Staubli VAL3: Sychron_slave.dtx

bool bCycleOn
bool bRb2Home
bool bRb2InitOk
bool bRb2Ready
bool bRealM
bool bRes
bool bSetIO = true
bool bSychronOn
public bool bTest = true
bool bTxt1
bool bTxt2
bool bTxt3
bool bTxtPrSv = true
public bool bfnshint
bool ststu
dio fOut0 = {link=fOut0}
frame FrmDraw = {x=627.549581, y=-600.363481, z=-159.173811, rx=-90.113097, ry=-0.047506, rz=-0.047357, fatherId=world[0]}
jointRx jCad = {j1=15.222913, j2=48.613048, j3=81.686613, j4=179.999698, j5=130.298951, j6=-15.223398}
jointRx jConfig = {j1=-56.268773, j2=69.307617, j3=102.367275, j4=127.245004, j5=114.935336, j6=-7.907875}
jointRx jHome = {j1=-56.268773, j2=69.307617, j3=102.367275, j4=127.245004, j5=114.935336, j6=-7.907875}
jointRx jReal = {j1=15.453516, j2=48.799216, j3=80.615756, j4=179.999705, j5=129.41426, j6=-15.453992}
public mdesc mNomSpeed = {accel=30, decel=30, tmax=600, rmax=600, blend=off}
mdesc mSlow = {accel=30, decel=30, tmax=500, rmax=500}
num CmdTotal
num nDbg
num nPtTotal = 5
num nPulse[1500]
  [0] = 1
  [2] = 1
  [4] = 1
  [6] = 1
  [8] = 1
  [10] = 1
  [12] = 1
  [14] = 1
  [16] = 1
  [18] = 1
  [20] = 1
  [22] = 1
  [24] = 1
  [26] = 1
  [28] = 1
  [30] = 1
  [32] = 1
  [34] = 1
  [36] = 1
  [38] = 1
  [40] = 1
  [42] = 1
  [44] = 1
  [46] = 1
  [48] = 1
  [50] = 1
  [52] = 1
  [54] = 1
  [56] = 1
  [58] = 1
  [60] = 1
  [62] = 1
  [64] = 1
  [66] = 1
  [68] = 1
  [70] = 1
  [72] = 1
  [74] = 1
  [76] = 1
  [78] = 1
  [80] = 1
  [82] = 1
  [84] = 1
  [86] = 1
  [88] = 1
  [90] = 1
  [92] = 1
  [94] = 1
  [96] = 1
  [98] = 1
  [100] = 1
  [102] = 1
  [104] = 1
  [106] = 1
  [108] = 1
  [110] = 1
  [112] = 1
  [114] = 1
  [116] = 1
  [118] = 1
  [120] = 1
  [122] = 1
  [124] = 1
  [126] = 1
  [128] = 1
  [130] = 1
  [132] = 1
  [134] = 1
  [136] = 1
  [138] = 1
  [140] = 1
  [142] = 1
  [144] = 1
  [146] = 1
  [148] = 1
  [150] = 1
  [152] = 1
  [154] = 1
  [156] = 1
  [158] = 1
  [160] = 1
  [162] = 1
  [164] = 1
  [166] = 1
  [168] = 1
  [170] = 1
  [172] = 1
  [174] = 1
  [176] = 1
  [178] = 1
  [180] = 1
  [182] = 1
  [184] = 1
  [186] = 1
  [188] = 1
  [190] = 1
  [192] = 1
  [194] = 1
  [196] = 1
  [198] = 1
  [200] = 1
  [202] = 1
  [204] = 1
  [206] = 1
  [208] = 1
  [210] = 1
  [212] = 1
  [214] = 1
  [216] = 1
  [218] = 1
  [220] = 1
  [222] = 1
  [224] = 1
  [226] = 1
  [228] = 1
  [230] = 1
  [232] = 1
  [234] = 1
  [236] = 1
  [238] = 1
  [240] = 1
  [242] = 1
  [244] = 1
  [246] = 1
  [248] = 1
  [250] = 1
  [252] = 1
  [254] = 1
  [256] = 1
  [258] = 1
  [260] = 1
  [262] = 1
  [264] = 1
  [266] = 1
  [268] = 1
  [270] = 1
  [272] = 1
  [274] = 1
  [276] = 1
  [278] = 1
  [280] = 1
  [282] = 1
  [284] = 1
  [286] = 1
  [288] = 1
  [290] = 1
  [292] = 1
  [294] = 1
  [296] = 1
  [298] = 1
  [300] = 1
  [302] = 1
  [304] = 1
  [306] = 1
  [308] = 1
  [310] = 1
  [312] = 1
  [314] = 1
  [316] = 1
  [318] = 1
  [320] = 1
  [322] = 1
  [324] = 1
  [326] = 1
  [328] = 1
  [330] = 1
  [332] = 1
  [334] = 1
  [336] = 1
  [338] = 1
  [340] = 1
  [342] = 1
  [344] = 1
  [346] = 1
  [348] = 1
  [350] = 1
  [352] = 1
  [354] = 1
  [356] = 1
  [358] = 1
  [360] = 1
  [362] = 1
  [364] = 1
  [366] = 1
  [368] = 1
  [370] = 1
  [372] = 1
  [374] = 1
  [376] = 1
  [378] = 1
  [380] = 1
  [382] = 1
  [384] = 1
  [386] = 1
  [388] = 1
  [390] = 1
  [392] = 1
  [394] = 1
  [396] = 1
  [398] = 1
  [400] = 1
  [402] = 1
  [404] = 1
  [406] = 1
  [408] = 1
  [410] = 1
  [412] = 1
  [414] = 1
  [416] = 1
  [418] = 1
  [420] = 1
  [422] = 1
  [424] = 1
  [426] = 1
  [428] = 1
  [430] = 1
  [432] = 1
  [434] = 1
  [436] = 1
  [438] = 1
  [440] = 1
  [442] = 1
  [444] = 1
  [446] = 1
  [448] = 1
  [450] = 1
  [452] = 1
  [454] = 1
  [456] = 1
  [458] = 1
  [460] = 1
  [462] = 1
  [464] = 1
  [466] = 1
  [468] = 1
  [470] = 1
  [472] = 1
  [474] = 1
  [476] = 1
  [478] = 1
  [480] = 1
  [482] = 1
  [484] = 1
  [486] = 1
  [488] = 1
  [490] = 1
  [492] = 1
  [494] = 1
  [496] = 1
  [498] = 1
  [500] = 1
  [502] = 1
  [504] = 1
  [506] = 1
  [508] = 1
  [510] = 1
  [512] = 1
  [514] = 1
  [516] = 1
  [518] = 1
  [520] = 1
  [522] = 1
  [524] = 1
  [526] = 1
  [528] = 1
  [530] = 1
  [532] = 1
  [534] = 1
  [536] = 1
  [538] = 1
  [540] = 1
  [542] = 1
  [544] = 1
  [546] = 1
  [548] = 1
  [550] = 1
  [552] = 1
  [554] = 1
  [556] = 1
  [558] = 1
  [560] = 1
  [562] = 1
  [564] = 1
  [566] = 1
  [568] = 1
  [570] = 1
  [572] = 1
  [574] = 1
  [576] = 1
  [578] = 1
  [580] = 1
  [582] = 1
  [584] = 1
  [586] = 1
  [588] = 1
  [590] = 1
  [592] = 1
  [594] = 1
  [596] = 1
  [598] = 1
  [600] = 1
  [602] = 1
  [604] = 1
  [606] = 1
  [608] = 1
  [610] = 1
  [612] = 1
  [614] = 1
  [616] = 1
  [618] = 1
  [620] = 1
  [622] = 1
  [624] = 1
  [626] = 1
  [628] = 1
  [630] = 1
  [632] = 1
  [634] = 1
  [636] = 1
  [638] = 1
  [640] = 1
  [642] = 1
  [644] = 1
  [646] = 1
  [648] = 1
  [650] = 1
  [652] = 1
  [654] = 1
  [656] = 1
  [658] = 1
  [660] = 1
  [662] = 1
  [664] = 1
  [666] = 1
  [668] = 1
  [670] = 1
  [672] = 1
  [674] = 1
  [676] = 1
  [678] = 1
  [680] = 1
  [682] = 1
  [684] = 1
  [686] = 1
  [688] = 1
  [690] = 1
  [692] = 1
  [694] = 1
  [696] = 1
  [698] = 1
  [700] = 1
  [702] = 1
  [704] = 1
  [706] = 1
  [708] = 1
  [710] = 1
  [712] = 1
  [714] = 1
  [716] = 1
  [718] = 1
  [720] = 1
  [722] = 1
  [724] = 1
  [726] = 1
  [728] = 1
  [730] = 1
  [732] = 1
  [734] = 1
  [736] = 1
  [738] = 1
  [740] = 1
  [742] = 1
  [744] = 1
  [746] = 1
  [748] = 1
  [750] = 1
  [752] = 1
  [754] = 1
  [756] = 1
  [758] = 1
  [760] = 1
  [762] = 1
  [764] = 1
  [766] = 1
  [768] = 1
  [770] = 1
  [772] = 1
  [774] = 1
  [776] = 1
  [778] = 1
  [780] = 1
  [782] = 1
  [784] = 1
  [786] = 1
  [788] = 1
  [790] = 1
  [792] = 1
  [794] = 1
  [796] = 1
  [798] = 1
  [800] = 1
  [802] = 1
  [804] = 1
  [806] = 1
  [808] = 1
  [810] = 1
  [812] = 1
  [814] = 1
  [816] = 1
  [818] = 1
  [820] = 1
  [822] = 1
  [824] = 1
  [826] = 1
  [828] = 1
  [830] = 1
  [832] = 1
  [834] = 1
  [836] = 1
  [838] = 1
  [840] = 1
  [842] = 1
  [844] = 1
  [846] = 1
  [848] = 1
  [850] = 1
  [852] = 1
  [854] = 1
  [856] = 1
  [858] = 1
  [860] = 1
  [862] = 1
  [864] = 1
  [866] = 1
  [868] = 1
  [870] = 1
  [872] = 1
  [874] = 1
  [876] = 1
  [878] = 1
  [880] = 1
  [882] = 1
  [884] = 1
  [886] = 1
  [888] = 1
  [890] = 1
  [892] = 1
  [894] = 1
  [896] = 1
  [898] = 1
  [900] = 1
  [902] = 1
  [904] = 1
  [906] = 1
  [908] = 1
  [910] = 1
  [912] = 1
  [914] = 1
  [916] = 1
  [918] = 1
  [920] = 1
  [922] = 1
  [924] = 1
  [926] = 1
  [928] = 1
  [930] = 1
  [932] = 1
  [934] = 1
  [936] = 1
  [938] = 1
  [940] = 1
  [942] = 1
  [944] = 1
  [946] = 1
  [948] = 1
  [950] = 1
  [952] = 1
  [954] = 1
  [956] = 1
  [958] = 1
  [960] = 1
  [962] = 1
  [964] = 1
  [966] = 1
  [968] = 1
  [970] = 1
  [972] = 1
  [974] = 1
  [976] = 1
  [978] = 1
  [980] = 1
  [982] = 1
  [984] = 1
  [986] = 1
  [988] = 1
  [990] = 1
  [992] = 1
  [994] = 1
  [996] = 1
  [998] = 1
num nReadPt
num nScrPts = 1291
public num nTestNum = 2
public num nTime = 0.001
num nTotalPoints = 1
num nTxtTotal = 347
num nWritePt
num n_sTxt = 2
num nn = 3048
num nsumtime = 5916.439
pointRx MoveTo = {ry=-90, rz=174.889504, fatherId=FrmDraw[0]}
pointRx Zero = {ry=-90, rz=174.889504, fatherId=FrmDraw[0]}
pointRx frm_ori = {x=627.549581, y=-600.363481, z=-159.173811, ry=90, rz=179.586129, fatherId=world[0]}
pointRx frm_x = {x=876.01171, y=-600.157069, z=-158.968855, rx=4.422019, ry=89.999088, rz=175.164786, fatherId=world[0]}
pointRx frm_y = {x=875.958066, y=-600.377284, z=-270.508394, ry=90, rz=179.586975, fatherId=world[0]}
pointRx pChange = {fatherId=FrmDraw[0]}
pointRx pfrmCad[1500]
  [0] = {x=52.63, y=-161.79, z=1, rx=-90, ry=53.98, fatherId=FrmDraw[0]}
  [1] = {x=52.51, y=-161.63, z=1, rx=-90, ry=54, fatherId=FrmDraw[0]}
  [2] = {x=52.39, y=-161.46, z=1, rx=-90, ry=54.05, fatherId=FrmDraw[0]}
  [3] = {x=52.27, y=-161.3, z=1, rx=-90, ry=54.09, fatherId=FrmDraw[0]}
  [4] = {x=52.16, y=-161.14, z=1, rx=-90, ry=54.13, fatherId=FrmDraw[0]}
  [5] = {x=52.04, y=-160.98, z=1, rx=-90, ry=54.17, fatherId=FrmDraw[0]}
  [6] = {x=51.92, y=-160.82, z=1, rx=-90, ry=54.21, fatherId=FrmDraw[0]}
  [7] = {x=51.81, y=-160.65, z=1, rx=-90, ry=54.25, fatherId=FrmDraw[0]}
  [8] = {x=51.69, y=-160.49, z=1, rx=-90, ry=54.3, fatherId=FrmDraw[0]}
  [9] = {x=51.57, y=-160.33, z=1, rx=-90, ry=54.34, fatherId=FrmDraw[0]}
  [10] = {x=51.46, y=-160.17, z=1, rx=-90, ry=54.38, fatherId=FrmDraw[0]}
  [11] = {x=51.34, y=-160, z=1, rx=-90, ry=54.42, fatherId=FrmDraw[0]}
  [12] = {x=51.22, y=-159.84, z=1, rx=-90, ry=54.46, fatherId=FrmDraw[0]}
  [13] = {x=51.11, y=-159.68, z=1, rx=-90, ry=54.5, fatherId=FrmDraw[0]}
  [14] = {x=50.99, y=-159.52, z=1, rx=-90, ry=54.55, fatherId=FrmDraw[0]}
  [15] = {x=50.88, y=-159.35, z=1, rx=-90, ry=54.59, fatherId=FrmDraw[0]}
  [16] = {x=50.76, y=-159.19, z=1, rx=-90, ry=54.63, fatherId=FrmDraw[0]}
  [17] = {x=50.64, y=-159.03, z=1, rx=-90, ry=54.67, fatherId=FrmDraw[0]}
  [18] = {x=50.53, y=-158.86, z=1, rx=-90, ry=54.71, fatherId=FrmDraw[0]}
  [19] = {x=50.41, y=-158.7, z=1, rx=-90, ry=54.75, fatherId=FrmDraw[0]}
  [20] = {x=50.3, y=-158.54, z=1, rx=-90, ry=54.8, fatherId=FrmDraw[0]}
  [21] = {x=50.18, y=-158.37, z=1, rx=-90, ry=54.84, fatherId=FrmDraw[0]}
  [22] = {x=50.07, y=-158.21, z=1, rx=-90, ry=54.88, fatherId=FrmDraw[0]}
  [23] = {x=49.95, y=-158.05, z=1, rx=-90, ry=54.92, fatherId=FrmDraw[0]}
  [24] = {x=49.84, y=-157.88, z=1, rx=-90, ry=54.96, fatherId=FrmDraw[0]}
  [25] = {x=49.72, y=-157.72, z=1, rx=-90, ry=55, fatherId=FrmDraw[0]}
  [26] = {x=49.61, y=-157.55, z=1, rx=-90, ry=55.05, fatherId=FrmDraw[0]}
  [27] = {x=49.49, y=-157.39, z=1, rx=-90, ry=55.09, fatherId=FrmDraw[0]}
  [28] = {x=49.38, y=-157.23, z=1, rx=-90, ry=55.13, fatherId=FrmDraw[0]}
  [29] = {x=49.26, y=-157.06, z=1, rx=-90, ry=55.17, fatherId=FrmDraw[0]}
  [30] = {x=49.15, y=-156.9, z=1, rx=-90, ry=55.21, fatherId=FrmDraw[0]}
  [31] = {x=49.04, y=-156.73, z=1, rx=-90, ry=55.25, fatherId=FrmDraw[0]}
  [32] = {x=48.92, y=-156.57, z=1, rx=-90, ry=55.3, fatherId=FrmDraw[0]}
  [33] = {x=48.81, y=-156.4, z=1, rx=-90, ry=55.34, fatherId=FrmDraw[0]}
  [34] = {x=48.69, y=-156.24, z=1, rx=-90, ry=55.38, fatherId=FrmDraw[0]}
  [35] = {x=48.58, y=-156.08, z=1, rx=-90, ry=55.42, fatherId=FrmDraw[0]}
  [36] = {x=48.47, y=-155.91, z=1, rx=-90, ry=55.46, fatherId=FrmDraw[0]}
  [37] = {x=48.35, y=-155.75, z=1, rx=-90, ry=55.5, fatherId=FrmDraw[0]}
  [38] = {x=48.24, y=-155.58, z=1, rx=-90, ry=55.55, fatherId=FrmDraw[0]}
  [39] = {x=48.13, y=-155.42, z=1, rx=-90, ry=55.59, fatherId=FrmDraw[0]}
  [40] = {x=48.02, y=-155.25, z=1, rx=-90, ry=55.63, fatherId=FrmDraw[0]}
  [41] = {x=47.9, y=-155.09, z=1, rx=-90, ry=55.67, fatherId=FrmDraw[0]}
  [42] = {x=47.79, y=-154.92, z=1, rx=-90, ry=55.71, fatherId=FrmDraw[0]}
  [43] = {x=47.68, y=-154.76, z=1, rx=-90, ry=55.75, fatherId=FrmDraw[0]}
  [44] = {x=47.56, y=-154.59, z=1, rx=-90, ry=55.8, fatherId=FrmDraw[0]}
  [45] = {x=47.45, y=-154.42, z=1, rx=-90, ry=55.84, fatherId=FrmDraw[0]}
  [46] = {x=47.34, y=-154.26, z=1, rx=-90, ry=55.88, fatherId=FrmDraw[0]}
  [47] = {x=47.23, y=-154.09, z=1, rx=-90, ry=55.92, fatherId=FrmDraw[0]}
  [48] = {x=47.12, y=-153.93, z=1, rx=-90, ry=55.96, fatherId=FrmDraw[0]}
  [49] = {x=47, y=-153.76, z=1, rx=-90, ry=56, fatherId=FrmDraw[0]}
  [50] = {x=46.89, y=-153.6, z=1, rx=-90, ry=56.05, fatherId=FrmDraw[0]}
  [51] = {x=46.78, y=-153.43, z=1, rx=-90, ry=56.09, fatherId=FrmDraw[0]}
  [52] = {x=46.67, y=-153.26, z=1, rx=-90, ry=56.13, fatherId=FrmDraw[0]}
  [53] = {x=46.56, y=-153.1, z=1, rx=-90, ry=56.17, fatherId=FrmDraw[0]}
  [54] = {x=46.45, y=-152.93, z=1, rx=-90, ry=56.21, fatherId=FrmDraw[0]}
  [55] = {x=46.34, y=-152.77, z=1, rx=-90, ry=56.25, fatherId=FrmDraw[0]}
  [56] = {x=46.22, y=-152.6, z=1, rx=-90, ry=56.3, fatherId=FrmDraw[0]}
  [57] = {x=46.11, y=-152.43, z=1, rx=-90, ry=56.34, fatherId=FrmDraw[0]}
  [58] = {x=46, y=-152.27, z=1, rx=-90, ry=56.38, fatherId=FrmDraw[0]}
  [59] = {x=45.89, y=-152.1, z=1, rx=-90, ry=56.42, fatherId=FrmDraw[0]}
  [60] = {x=45.78, y=-151.93, z=1, rx=-90, ry=56.46, fatherId=FrmDraw[0]}
  [61] = {x=45.67, y=-151.77, z=1, rx=-90, ry=56.5, fatherId=FrmDraw[0]}
  [62] = {x=45.56, y=-151.6, z=1, rx=-90, ry=56.55, fatherId=FrmDraw[0]}
  [63] = {x=45.45, y=-151.43, z=1, rx=-90, ry=56.59, fatherId=FrmDraw[0]}
  [64] = {x=45.34, y=-151.27, z=1, rx=-90, ry=56.63, fatherId=FrmDraw[0]}
  [65] = {x=45.23, y=-151.1, z=1, rx=-90, ry=56.67, fatherId=FrmDraw[0]}
  [66] = {x=45.12, y=-150.93, z=1, rx=-90, ry=56.71, fatherId=FrmDraw[0]}
  [67] = {x=45.01, y=-150.76, z=1, rx=-90, ry=56.75, fatherId=FrmDraw[0]}
  [68] = {x=44.9, y=-150.6, z=1, rx=-90, ry=56.8, fatherId=FrmDraw[0]}
  [69] = {x=44.79, y=-150.43, z=1, rx=-90, ry=56.84, fatherId=FrmDraw[0]}
  [70] = {x=44.68, y=-150.26, z=1, rx=-90, ry=56.88, fatherId=FrmDraw[0]}
  [71] = {x=44.57, y=-150.09, z=1, rx=-90, ry=56.92, fatherId=FrmDraw[0]}
  [72] = {x=44.46, y=-149.93, z=1, rx=-90, ry=56.96, fatherId=FrmDraw[0]}
  [73] = {x=44.35, y=-149.76, z=1, rx=-90, ry=57, fatherId=FrmDraw[0]}
  [74] = {x=44.25, y=-149.59, z=1, rx=-90, ry=57.05, fatherId=FrmDraw[0]}
  [75] = {x=44.14, y=-149.42, z=1, rx=-90, ry=57.09, fatherId=FrmDraw[0]}
  [76] = {x=44.03, y=-149.26, z=1, rx=-90, ry=57.13, fatherId=FrmDraw[0]}
  [77] = {x=43.92, y=-149.09, z=1, rx=-90, ry=57.17, fatherId=FrmDraw[0]}
  [78] = {x=43.81, y=-148.92, z=1, rx=-90, ry=57.21, fatherId=FrmDraw[0]}
  [79] = {x=43.7, y=-148.75, z=1, rx=-90, ry=57.25, fatherId=FrmDraw[0]}
  [80] = {x=43.6, y=-148.58, z=1, rx=-90, ry=57.3, fatherId=FrmDraw[0]}
  [81] = {x=43.49, y=-148.41, z=1, rx=-90, ry=57.34, fatherId=FrmDraw[0]}
  [82] = {x=43.38, y=-148.25, z=1, rx=-90, ry=57.38, fatherId=FrmDraw[0]}
  [83] = {x=43.27, y=-148.08, z=1, rx=-90, ry=57.42, fatherId=FrmDraw[0]}
  [84] = {x=43.16, y=-147.91, z=1, rx=-90, ry=57.46, fatherId=FrmDraw[0]}
  [85] = {x=43.06, y=-147.74, z=1, rx=-90, ry=57.5, fatherId=FrmDraw[0]}
  [86] = {x=42.95, y=-147.57, z=1, rx=-90, ry=57.55, fatherId=FrmDraw[0]}
  [87] = {x=42.84, y=-147.4, z=1, rx=-90, ry=57.59, fatherId=FrmDraw[0]}
  [88] = {x=42.73, y=-147.23, z=1, rx=-90, ry=57.63, fatherId=FrmDraw[0]}
  [89] = {x=42.63, y=-147.07, z=1, rx=-90, ry=57.67, fatherId=FrmDraw[0]}
  [90] = {x=42.52, y=-146.9, z=1, rx=-90, ry=57.71, fatherId=FrmDraw[0]}
  [91] = {x=42.41, y=-146.73, z=1, rx=-90, ry=57.75, fatherId=FrmDraw[0]}
  [92] = {x=42.31, y=-146.56, z=1, rx=-90, ry=57.8, fatherId=FrmDraw[0]}
  [93] = {x=42.2, y=-146.39, z=1, rx=-90, ry=57.84, fatherId=FrmDraw[0]}
  [94] = {x=42.09, y=-146.22, z=1, rx=-90, ry=57.88, fatherId=FrmDraw[0]}
  [95] = {x=41.99, y=-146.05, z=1, rx=-90, ry=57.92, fatherId=FrmDraw[0]}
  [96] = {x=41.88, y=-145.88, z=1, rx=-90, ry=57.96, fatherId=FrmDraw[0]}
  [97] = {x=41.78, y=-145.71, z=1, rx=-90, ry=58, fatherId=FrmDraw[0]}
  [98] = {x=41.67, y=-145.54, z=1, rx=-90, ry=58.05, fatherId=FrmDraw[0]}
  [99] = {x=41.56, y=-145.37, z=1, rx=-90, ry=58.09, fatherId=FrmDraw[0]}
  [100] = {x=41.46, y=-145.2, z=1, rx=-90, ry=58.13, fatherId=FrmDraw[0]}
  [101] = {x=41.35, y=-145.03, z=1, rx=-90, ry=58.17, fatherId=FrmDraw[0]}
  [102] = {x=41.25, y=-144.86, z=1, rx=-90, ry=58.21, fatherId=FrmDraw[0]}
  [103] = {x=41.14, y=-144.69, z=1, rx=-90, ry=58.25, fatherId=FrmDraw[0]}
  [104] = {x=41.04, y=-144.52, z=1, rx=-90, ry=58.3, fatherId=FrmDraw[0]}
  [105] = {x=40.93, y=-144.35, z=1, rx=-90, ry=58.34, fatherId=FrmDraw[0]}
  [106] = {x=40.83, y=-144.18, z=1, rx=-90, ry=58.38, fatherId=FrmDraw[0]}
  [107] = {x=40.72, y=-144.01, z=1, rx=-90, ry=58.42, fatherId=FrmDraw[0]}
  [108] = {x=40.62, y=-143.84, z=1, rx=-90, ry=58.46, fatherId=FrmDraw[0]}
  [109] = {x=40.51, y=-143.67, z=1, rx=-90, ry=58.5, fatherId=FrmDraw[0]}
  [110] = {x=40.41, y=-143.5, z=1, rx=-90, ry=58.55, fatherId=FrmDraw[0]}
  [111] = {x=40.3, y=-143.33, z=1, rx=-90, ry=58.59, fatherId=FrmDraw[0]}
  [112] = {x=40.2, y=-143.16, z=1, rx=-90, ry=58.63, fatherId=FrmDraw[0]}
  [113] = {x=40.1, y=-142.99, z=1, rx=-90, ry=58.67, fatherId=FrmDraw[0]}
  [114] = {x=39.99, y=-142.82, z=1, rx=-90, ry=58.71, fatherId=FrmDraw[0]}
  [115] = {x=39.89, y=-142.65, z=1, rx=-90, ry=58.75, fatherId=FrmDraw[0]}
  [116] = {x=39.79, y=-142.47, z=1, rx=-90, ry=58.8, fatherId=FrmDraw[0]}
  [117] = {x=39.68, y=-142.3, z=1, rx=-90, ry=58.84, fatherId=FrmDraw[0]}
  [118] = {x=39.58, y=-142.13, z=1, rx=-90, ry=58.88, fatherId=FrmDraw[0]}
  [119] = {x=39.47, y=-141.96, z=1, rx=-90, ry=58.92, fatherId=FrmDraw[0]}
  [120] = {x=39.37, y=-141.79, z=1, rx=-90, ry=58.96, fatherId=FrmDraw[0]}
  [121] = {x=39.27, y=-141.62, z=1, rx=-90, ry=59, fatherId=FrmDraw[0]}
  [122] = {x=39.17, y=-141.45, z=1, rx=-90, ry=59.05, fatherId=FrmDraw[0]}
  [123] = {x=39.06, y=-141.28, z=1, rx=-90, ry=59.09, fatherId=FrmDraw[0]}
  [124] = {x=38.96, y=-141.1, z=1, rx=-90, ry=59.13, fatherId=FrmDraw[0]}
  [125] = {x=38.86, y=-140.93, z=1, rx=-90, ry=59.17, fatherId=FrmDraw[0]}
  [126] = {x=38.76, y=-140.76, z=1, rx=-90, ry=59.21, fatherId=FrmDraw[0]}
  [127] = {x=38.65, y=-140.59, z=1, rx=-90, ry=59.25, fatherId=FrmDraw[0]}
  [128] = {x=38.55, y=-140.42, z=1, rx=-90, ry=59.3, fatherId=FrmDraw[0]}
  [129] = {x=38.45, y=-140.24, z=1, rx=-90, ry=59.34, fatherId=FrmDraw[0]}
  [130] = {x=38.35, y=-140.07, z=1, rx=-90, ry=59.38, fatherId=FrmDraw[0]}
  [131] = {x=38.24, y=-139.9, z=1, rx=-90, ry=59.42, fatherId=FrmDraw[0]}
  [132] = {x=38.14, y=-139.73, z=1, rx=-90, ry=59.46, fatherId=FrmDraw[0]}
  [133] = {x=38.04, y=-139.56, z=1, rx=-90, ry=59.5, fatherId=FrmDraw[0]}
  [134] = {x=37.94, y=-139.38, z=1, rx=-90, ry=59.55, fatherId=FrmDraw[0]}
  [135] = {x=37.84, y=-139.21, z=1, rx=-90, ry=59.59, fatherId=FrmDraw[0]}
  [136] = {x=37.74, y=-139.04, z=1, rx=-90, ry=59.63, fatherId=FrmDraw[0]}
  [137] = {x=37.64, y=-138.87, z=1, rx=-90, ry=59.67, fatherId=FrmDraw[0]}
  [138] = {x=37.54, y=-138.69, z=1, rx=-90, ry=59.71, fatherId=FrmDraw[0]}
  [139] = {x=37.43, y=-138.52, z=1, rx=-90, ry=59.75, fatherId=FrmDraw[0]}
  [140] = {x=37.33, y=-138.35, z=1, rx=-90, ry=59.8, fatherId=FrmDraw[0]}
  [141] = {x=37.23, y=-138.17, z=1, rx=-90, ry=59.84, fatherId=FrmDraw[0]}
  [142] = {x=37.13, y=-138, z=1, rx=-90, ry=59.88, fatherId=FrmDraw[0]}
  [143] = {x=37.03, y=-137.83, z=1, rx=-90, ry=59.92, fatherId=FrmDraw[0]}
  [144] = {x=36.93, y=-137.66, z=1, rx=-90, ry=59.96, fatherId=FrmDraw[0]}
  [145] = {x=36.83, y=-137.48, z=1, rx=-90, ry=60, fatherId=FrmDraw[0]}
  [146] = {x=36.73, y=-137.31, z=1, rx=-90, ry=60.05, fatherId=FrmDraw[0]}
  [147] = {x=36.63, y=-137.14, z=1, rx=-90, ry=60.09, fatherId=FrmDraw[0]}
  [148] = {x=36.53, y=-136.96, z=1, rx=-90, ry=60.13, fatherId=FrmDraw[0]}
  [149] = {x=36.43, y=-136.79, z=1, rx=-90, ry=60.17, fatherId=FrmDraw[0]}
  [150] = {x=36.33, y=-136.62, z=1, rx=-90, ry=60.21, fatherId=FrmDraw[0]}
  [151] = {x=36.24, y=-136.44, z=1, rx=-90, ry=60.25, fatherId=FrmDraw[0]}
  [152] = {x=36.14, y=-136.27, z=1, rx=-90, ry=60.3, fatherId=FrmDraw[0]}
  [153] = {x=36.04, y=-136.09, z=1, rx=-90, ry=60.34, fatherId=FrmDraw[0]}
  [154] = {x=35.94, y=-135.92, z=1, rx=-90, ry=60.38, fatherId=FrmDraw[0]}
  [155] = {x=35.84, y=-135.75, z=1, rx=-90, ry=60.42, fatherId=FrmDraw[0]}
  [156] = {x=35.74, y=-135.57, z=1, rx=-90, ry=60.46, fatherId=FrmDraw[0]}
  [157] = {x=35.64, y=-135.4, z=1, rx=-90, ry=60.5, fatherId=FrmDraw[0]}
  [158] = {x=35.54, y=-135.22, z=1, rx=-90, ry=60.55, fatherId=FrmDraw[0]}
  [159] = {x=35.45, y=-135.05, z=1, rx=-90, ry=60.59, fatherId=FrmDraw[0]}
  [160] = {x=35.35, y=-134.88, z=1, rx=-90, ry=60.63, fatherId=FrmDraw[0]}
  [161] = {x=35.25, y=-134.7, z=1, rx=-90, ry=60.67, fatherId=FrmDraw[0]}
  [162] = {x=35.15, y=-134.53, z=1, rx=-90, ry=60.71, fatherId=FrmDraw[0]}
  [163] = {x=35.05, y=-134.35, z=1, rx=-90, ry=60.75, fatherId=FrmDraw[0]}
  [164] = {x=34.96, y=-134.18, z=1, rx=-90, ry=60.8, fatherId=FrmDraw[0]}
  [165] = {x=34.86, y=-134, z=1, rx=-90, ry=60.84, fatherId=FrmDraw[0]}
  [166] = {x=34.76, y=-133.83, z=1, rx=-90, ry=60.88, fatherId=FrmDraw[0]}
  [167] = {x=34.66, y=-133.65, z=1, rx=-90, ry=60.92, fatherId=FrmDraw[0]}
  [168] = {x=34.57, y=-133.48, z=1, rx=-90, ry=60.96, fatherId=FrmDraw[0]}
  [169] = {x=34.47, y=-133.3, z=1, rx=-90, ry=61, fatherId=FrmDraw[0]}
  [170] = {x=34.37, y=-133.13, z=1, rx=-90, ry=61.05, fatherId=FrmDraw[0]}
  [171] = {x=34.28, y=-132.95, z=1, rx=-90, ry=61.09, fatherId=FrmDraw[0]}
  [172] = {x=34.18, y=-132.78, z=1, rx=-90, ry=61.13, fatherId=FrmDraw[0]}
  [173] = {x=34.08, y=-132.6, z=1, rx=-90, ry=61.17, fatherId=FrmDraw[0]}
  [174] = {x=33.99, y=-132.43, z=1, rx=-90, ry=61.21, fatherId=FrmDraw[0]}
  [175] = {x=33.89, y=-132.25, z=1, rx=-90, ry=61.25, fatherId=FrmDraw[0]}
  [176] = {x=33.79, y=-132.08, z=1, rx=-90, ry=61.3, fatherId=FrmDraw[0]}
  [177] = {x=33.7, y=-131.9, z=1, rx=-90, ry=61.34, fatherId=FrmDraw[0]}
  [178] = {x=33.6, y=-131.73, z=1, rx=-90, ry=61.38, fatherId=FrmDraw[0]}
  [179] = {x=33.51, y=-131.55, z=1, rx=-90, ry=61.42, fatherId=FrmDraw[0]}
  [180] = {x=33.41, y=-131.38, z=1, rx=-90, ry=61.46, fatherId=FrmDraw[0]}
  [181] = {x=33.32, y=-131.2, z=1, rx=-90, ry=61.5, fatherId=FrmDraw[0]}
  [182] = {x=33.22, y=-131.02, z=1, rx=-90, ry=61.55, fatherId=FrmDraw[0]}
  [183] = {x=33.12, y=-130.85, z=1, rx=-90, ry=61.59, fatherId=FrmDraw[0]}
  [184] = {x=33.03, y=-130.67, z=1, rx=-90, ry=61.63, fatherId=FrmDraw[0]}
  [185] = {x=32.93, y=-130.5, z=1, rx=-90, ry=61.67, fatherId=FrmDraw[0]}
  [186] = {x=32.84, y=-130.32, z=1, rx=-90, ry=61.71, fatherId=FrmDraw[0]}
  [187] = {x=32.74, y=-130.14, z=1, rx=-90, ry=61.75, fatherId=FrmDraw[0]}
  [188] = {x=32.65, y=-129.97, z=1, rx=-90, ry=61.8, fatherId=FrmDraw[0]}
  [189] = {x=32.56, y=-129.79, z=1, rx=-90, ry=61.84, fatherId=FrmDraw[0]}
  [190] = {x=32.46, y=-129.62, z=1, rx=-90, ry=61.88, fatherId=FrmDraw[0]}
  [191] = {x=32.37, y=-129.44, z=1, rx=-90, ry=61.92, fatherId=FrmDraw[0]}
  [192] = {x=32.27, y=-129.26, z=1, rx=-90, ry=61.96, fatherId=FrmDraw[0]}
  [193] = {x=32.18, y=-129.09, z=1, rx=-90, ry=62, fatherId=FrmDraw[0]}
  [194] = {x=32.09, y=-128.91, z=1, rx=-90, ry=62.05, fatherId=FrmDraw[0]}
  [195] = {x=31.99, y=-128.73, z=1, rx=-90, ry=62.09, fatherId=FrmDraw[0]}
  [196] = {x=31.9, y=-128.56, z=1, rx=-90, ry=62.13, fatherId=FrmDraw[0]}
  [197] = {x=31.8, y=-128.38, z=1, rx=-90, ry=62.17, fatherId=FrmDraw[0]}
  [198] = {x=31.71, y=-128.2, z=1, rx=-90, ry=62.21, fatherId=FrmDraw[0]}
  [199] = {x=31.62, y=-128.03, z=1, rx=-90, ry=62.25, fatherId=FrmDraw[0]}
  [200] = {x=31.53, y=-127.85, z=1, rx=-90, ry=62.3, fatherId=FrmDraw[0]}
  [201] = {x=31.43, y=-127.67, z=1, rx=-90, ry=62.34, fatherId=FrmDraw[0]}
  [202] = {x=31.34, y=-127.49, z=1, rx=-90, ry=62.38, fatherId=FrmDraw[0]}
  [203] = {x=31.25, y=-127.32, z=1, rx=-90, ry=62.42, fatherId=FrmDraw[0]}
  [204] = {x=31.15, y=-127.14, z=1, rx=-90, ry=62.46, fatherId=FrmDraw[0]}
  [205] = {x=31.06, y=-126.96, z=1, rx=-90, ry=62.5, fatherId=FrmDraw[0]}
  [206] = {x=30.97, y=-126.78, z=1, rx=-90, ry=62.55, fatherId=FrmDraw[0]}
  [207] = {x=30.88, y=-126.61, z=1, rx=-90, ry=62.59, fatherId=FrmDraw[0]}
  [208] = {x=30.79, y=-126.43, z=1, rx=-90, ry=62.63, fatherId=FrmDraw[0]}
  [209] = {x=30.69, y=-126.25, z=1, rx=-90, ry=62.67, fatherId=FrmDraw[0]}
  [210] = {x=30.6, y=-126.07, z=1, rx=-90, ry=62.71, fatherId=FrmDraw[0]}
  [211] = {x=30.51, y=-125.9, z=1, rx=-90, ry=62.75, fatherId=FrmDraw[0]}
  [212] = {x=30.42, y=-125.72, z=1, rx=-90, ry=62.8, fatherId=FrmDraw[0]}
  [213] = {x=30.33, y=-125.54, z=1, rx=-90, ry=62.84, fatherId=FrmDraw[0]}
  [214] = {x=30.24, y=-125.36, z=1, rx=-90, ry=62.88, fatherId=FrmDraw[0]}
  [215] = {x=30.15, y=-125.18, z=1, rx=-90, ry=62.92, fatherId=FrmDraw[0]}
  [216] = {x=30.05, y=-125.01, z=1, rx=-90, ry=62.96, fatherId=FrmDraw[0]}
  [217] = {x=29.96, y=-124.83, z=1, rx=-90, ry=63, fatherId=FrmDraw[0]}
  [218] = {x=29.87, y=-124.65, z=1, rx=-90, ry=63.05, fatherId=FrmDraw[0]}
  [219] = {x=29.78, y=-124.47, z=1, rx=-90, ry=63.09, fatherId=FrmDraw[0]}
  [220] = {x=29.69, y=-124.29, z=1, rx=-90, ry=63.13, fatherId=FrmDraw[0]}
  [221] = {x=29.6, y=-124.11, z=1, rx=-90, ry=63.17, fatherId=FrmDraw[0]}
  [222] = {x=29.51, y=-123.94, z=1, rx=-90, ry=63.21, fatherId=FrmDraw[0]}
  [223] = {x=29.42, y=-123.76, z=1, rx=-90, ry=63.25, fatherId=FrmDraw[0]}
  [224] = {x=29.33, y=-123.58, z=1, rx=-90, ry=63.3, fatherId=FrmDraw[0]}
  [225] = {x=29.24, y=-123.4, z=1, rx=-90, ry=63.34, fatherId=FrmDraw[0]}
  [226] = {x=29.15, y=-123.22, z=1, rx=-90, ry=63.38, fatherId=FrmDraw[0]}
  [227] = {x=29.06, y=-123.04, z=1, rx=-90, ry=63.42, fatherId=FrmDraw[0]}
  [228] = {x=28.97, y=-122.86, z=1, rx=-90, ry=63.46, fatherId=FrmDraw[0]}
  [229] = {x=28.88, y=-122.68, z=1, rx=-90, ry=63.5, fatherId=FrmDraw[0]}
  [230] = {x=28.79, y=-122.51, z=1, rx=-90, ry=63.55, fatherId=FrmDraw[0]}
  [231] = {x=28.71, y=-122.33, z=1, rx=-90, ry=63.59, fatherId=FrmDraw[0]}
  [232] = {x=28.62, y=-122.15, z=1, rx=-90, ry=63.63, fatherId=FrmDraw[0]}
  [233] = {x=28.53, y=-121.97, z=1, rx=-90, ry=63.67, fatherId=FrmDraw[0]}
  [234] = {x=28.44, y=-121.79, z=1, rx=-90, ry=63.71, fatherId=FrmDraw[0]}
  [235] = {x=28.35, y=-121.61, z=1, rx=-90, ry=63.75, fatherId=FrmDraw[0]}
  [236] = {x=28.26, y=-121.43, z=1, rx=-90, ry=63.8, fatherId=FrmDraw[0]}
  [237] = {x=28.17, y=-121.25, z=1, rx=-90, ry=63.84, fatherId=FrmDraw[0]}
  [238] = {x=28.09, y=-121.07, z=1, rx=-90, ry=63.88, fatherId=FrmDraw[0]}
  [239] = {x=28, y=-120.89, z=1, rx=-90, ry=63.92, fatherId=FrmDraw[0]}
  [240] = {x=27.91, y=-120.71, z=1, rx=-90, ry=63.96, fatherId=FrmDraw[0]}
  [241] = {x=27.82, y=-120.53, z=1, rx=-90, ry=64, fatherId=FrmDraw[0]}
  [242] = {x=27.73, y=-120.35, z=1, rx=-90, ry=64.05, fatherId=FrmDraw[0]}
  [243] = {x=27.65, y=-120.17, z=1, rx=-90, ry=64.09, fatherId=FrmDraw[0]}
  [244] = {x=27.56, y=-119.99, z=1, rx=-90, ry=64.13, fatherId=FrmDraw[0]}
  [245] = {x=27.47, y=-119.81, z=1, rx=-90, ry=64.17, fatherId=FrmDraw[0]}
  [246] = {x=27.39, y=-119.63, z=1, rx=-90, ry=64.21, fatherId=FrmDraw[0]}
  [247] = {x=27.3, y=-119.45, z=1, rx=-90, ry=64.25, fatherId=FrmDraw[0]}
  [248] = {x=27.21, y=-119.27, z=1, rx=-90, ry=64.3, fatherId=FrmDraw[0]}
  [249] = {x=27.12, y=-119.09, z=1, rx=-90, ry=64.34, fatherId=FrmDraw[0]}
  [250] = {x=27.04, y=-118.91, z=1, rx=-90, ry=64.38, fatherId=FrmDraw[0]}
  [251] = {x=26.95, y=-118.73, z=1, rx=-90, ry=64.42, fatherId=FrmDraw[0]}
  [252] = {x=26.87, y=-118.55, z=1, rx=-90, ry=64.46, fatherId=FrmDraw[0]}
  [253] = {x=26.78, y=-118.37, z=1, rx=-90, ry=64.5, fatherId=FrmDraw[0]}
  [254] = {x=26.69, y=-118.19, z=1, rx=-90, ry=64.55, fatherId=FrmDraw[0]}
  [255] = {x=26.61, y=-118.01, z=1, rx=-90, ry=64.59, fatherId=FrmDraw[0]}
  [256] = {x=26.52, y=-117.83, z=1, rx=-90, ry=64.63, fatherId=FrmDraw[0]}
  [257] = {x=26.44, y=-117.65, z=1, rx=-90, ry=64.67, fatherId=FrmDraw[0]}
  [258] = {x=26.35, y=-117.47, z=1, rx=-90, ry=64.71, fatherId=FrmDraw[0]}
  [259] = {x=26.27, y=-117.29, z=1, rx=-90, ry=64.75, fatherId=FrmDraw[0]}
  [260] = {x=26.18, y=-117.11, z=1, rx=-90, ry=64.8, fatherId=FrmDraw[0]}
  [261] = {x=26.09, y=-116.92, z=1, rx=-90, ry=64.84, fatherId=FrmDraw[0]}
  [262] = {x=26.01, y=-116.74, z=1, rx=-90, ry=64.88, fatherId=FrmDraw[0]}
  [263] = {x=25.93, y=-116.56, z=1, rx=-90, ry=64.92, fatherId=FrmDraw[0]}
  [264] = {x=25.84, y=-116.38, z=1, rx=-90, ry=64.96, fatherId=FrmDraw[0]}
  [265] = {x=25.76, y=-116.2, z=1, rx=-90, ry=65, fatherId=FrmDraw[0]}
  [266] = {x=25.67, y=-116.02, z=1, rx=-90, ry=65.05, fatherId=FrmDraw[0]}
  [267] = {x=25.59, y=-115.84, z=1, rx=-90, ry=65.09, fatherId=FrmDraw[0]}
  [268] = {x=25.5, y=-115.66, z=1, rx=-90, ry=65.13, fatherId=FrmDraw[0]}
  [269] = {x=25.42, y=-115.47, z=1, rx=-90, ry=65.17, fatherId=FrmDraw[0]}
  [270] = {x=25.33, y=-115.29, z=1, rx=-90, ry=65.21, fatherId=FrmDraw[0]}
  [271] = {x=25.25, y=-115.11, z=1, rx=-90, ry=65.25, fatherId=FrmDraw[0]}
  [272] = {x=25.17, y=-114.93, z=1, rx=-90, ry=65.3, fatherId=FrmDraw[0]}
  [273] = {x=25.08, y=-114.75, z=1, rx=-90, ry=65.34, fatherId=FrmDraw[0]}
  [274] = {x=25, y=-114.57, z=1, rx=-90, ry=65.38, fatherId=FrmDraw[0]}
  [275] = {x=24.92, y=-114.38, z=1, rx=-90, ry=65.42, fatherId=FrmDraw[0]}
  [276] = {x=24.83, y=-114.2, z=1, rx=-90, ry=65.46, fatherId=FrmDraw[0]}
  [277] = {x=24.75, y=-114.02, z=1, rx=-90, ry=65.5, fatherId=FrmDraw[0]}
  [278] = {x=24.67, y=-113.84, z=1, rx=-90, ry=65.55, fatherId=FrmDraw[0]}
  [279] = {x=24.59, y=-113.66, z=1, rx=-90, ry=65.59, fatherId=FrmDraw[0]}
  [280] = {x=24.5, y=-113.47, z=1, rx=-90, ry=65.63, fatherId=FrmDraw[0]}
  [281] = {x=24.42, y=-113.29, z=1, rx=-90, ry=65.67, fatherId=FrmDraw[0]}
  [282] = {x=24.34, y=-113.11, z=1, rx=-90, ry=65.71, fatherId=FrmDraw[0]}
  [283] = {x=24.26, y=-112.93, z=1, rx=-90, ry=65.75, fatherId=FrmDraw[0]}
  [284] = {x=24.17, y=-112.74, z=1, rx=-90, ry=65.8, fatherId=FrmDraw[0]}
  [285] = {x=24.09, y=-112.56, z=1, rx=-90, ry=65.84, fatherId=FrmDraw[0]}
  [286] = {x=24.01, y=-112.38, z=1, rx=-90, ry=65.88, fatherId=FrmDraw[0]}
  [287] = {x=23.93, y=-112.2, z=1, rx=-90, ry=65.92, fatherId=FrmDraw[0]}
  [288] = {x=23.85, y=-112.01, z=1, rx=-90, ry=65.96, fatherId=FrmDraw[0]}
  [289] = {x=23.77, y=-111.83, z=1, rx=-90, ry=66, fatherId=FrmDraw[0]}
  [290] = {x=23.68, y=-111.65, z=1, rx=-90, ry=66.05, fatherId=FrmDraw[0]}
  [291] = {x=23.6, y=-111.47, z=1, rx=-90, ry=66.09, fatherId=FrmDraw[0]}
  [292] = {x=23.52, y=-111.28, z=1, rx=-90, ry=66.13, fatherId=FrmDraw[0]}
  [293] = {x=23.44, y=-111.1, z=1, rx=-90, ry=66.17, fatherId=FrmDraw[0]}
  [294] = {x=23.36, y=-110.92, z=1, rx=-90, ry=66.21, fatherId=FrmDraw[0]}
  [295] = {x=23.28, y=-110.73, z=1, rx=-90, ry=66.25, fatherId=FrmDraw[0]}
  [296] = {x=23.2, y=-110.55, z=1, rx=-90, ry=66.3, fatherId=FrmDraw[0]}
  [297] = {x=23.12, y=-110.37, z=1, rx=-90, ry=66.34, fatherId=FrmDraw[0]}
  [298] = {x=23.04, y=-110.18, z=1, rx=-90, ry=66.38, fatherId=FrmDraw[0]}
  [299] = {x=22.96, y=-110, z=1, rx=-90, ry=66.42, fatherId=FrmDraw[0]}
  [300] = {x=22.88, y=-109.82, z=1, rx=-90, ry=66.46, fatherId=FrmDraw[0]}
  [301] = {x=22.8, y=-109.63, z=1, rx=-90, ry=66.5, fatherId=FrmDraw[0]}
  [302] = {x=22.72, y=-109.45, z=1, rx=-90, ry=66.55, fatherId=FrmDraw[0]}
  [303] = {x=22.64, y=-109.27, z=1, rx=-90, ry=66.59, fatherId=FrmDraw[0]}
  [304] = {x=22.56, y=-109.08, z=1, rx=-90, ry=66.63, fatherId=FrmDraw[0]}
  [305] = {x=22.48, y=-108.9, z=1, rx=-90, ry=66.67, fatherId=FrmDraw[0]}
  [306] = {x=22.4, y=-108.72, z=1, rx=-90, ry=66.71, fatherId=FrmDraw[0]}
  [307] = {x=22.32, y=-108.53, z=1, rx=-90, ry=66.75, fatherId=FrmDraw[0]}
  [308] = {x=22.24, y=-108.35, z=1, rx=-90, ry=66.8, fatherId=FrmDraw[0]}
  [309] = {x=22.17, y=-108.17, z=1, rx=-90, ry=66.84, fatherId=FrmDraw[0]}
  [310] = {x=22.09, y=-107.98, z=1, rx=-90, ry=66.88, fatherId=FrmDraw[0]}
  [311] = {x=22.01, y=-107.8, z=1, rx=-90, ry=66.92, fatherId=FrmDraw[0]}
  [312] = {x=21.93, y=-107.61, z=1, rx=-90, ry=66.96, fatherId=FrmDraw[0]}
  [313] = {x=21.85, y=-107.43, z=1, rx=-90, ry=67, fatherId=FrmDraw[0]}
  [314] = {x=21.77, y=-107.25, z=1, rx=-90, ry=67.05, fatherId=FrmDraw[0]}
  [315] = {x=21.7, y=-107.06, z=1, rx=-90, ry=67.09, fatherId=FrmDraw[0]}
  [316] = {x=21.62, y=-106.88, z=1, rx=-90, ry=67.13, fatherId=FrmDraw[0]}
  [317] = {x=21.54, y=-106.69, z=1, rx=-90, ry=67.17, fatherId=FrmDraw[0]}
  [318] = {x=21.46, y=-106.51, z=1, rx=-90, ry=67.21, fatherId=FrmDraw[0]}
  [319] = {x=21.39, y=-106.32, z=1, rx=-90, ry=67.25, fatherId=FrmDraw[0]}
  [320] = {x=21.31, y=-106.14, z=1, rx=-90, ry=67.3, fatherId=FrmDraw[0]}
  [321] = {x=21.23, y=-105.96, z=1, rx=-90, ry=67.34, fatherId=FrmDraw[0]}
  [322] = {x=21.15, y=-105.77, z=1, rx=-90, ry=67.38, fatherId=FrmDraw[0]}
  [323] = {x=21.08, y=-105.59, z=1, rx=-90, ry=67.42, fatherId=FrmDraw[0]}
  [324] = {x=21, y=-105.4, z=1, rx=-90, ry=67.46, fatherId=FrmDraw[0]}
  [325] = {x=20.92, y=-105.22, z=1, rx=-90, ry=67.5, fatherId=FrmDraw[0]}
  [326] = {x=20.85, y=-105.03, z=1, rx=-90, ry=67.55, fatherId=FrmDraw[0]}
  [327] = {x=20.77, y=-104.85, z=1, rx=-90, ry=67.59, fatherId=FrmDraw[0]}
  [328] = {x=20.7, y=-104.66, z=1, rx=-90, ry=67.63, fatherId=FrmDraw[0]}
  [329] = {x=20.62, y=-104.48, z=1, rx=-90, ry=67.67, fatherId=FrmDraw[0]}
  [330] = {x=20.54, y=-104.29, z=1, rx=-90, ry=67.71, fatherId=FrmDraw[0]}
  [331] = {x=20.47, y=-104.11, z=1, rx=-90, ry=67.75, fatherId=FrmDraw[0]}
  [332] = {x=20.39, y=-103.92, z=1, rx=-90, ry=67.8, fatherId=FrmDraw[0]}
  [333] = {x=20.32, y=-103.74, z=1, rx=-90, ry=67.84, fatherId=FrmDraw[0]}
  [334] = {x=20.24, y=-103.55, z=1, rx=-90, ry=67.88, fatherId=FrmDraw[0]}
  [335] = {x=20.17, y=-103.37, z=1, rx=-90, ry=67.92, fatherId=FrmDraw[0]}
  [336] = {x=20.09, y=-103.18, z=1, rx=-90, ry=67.96, fatherId=FrmDraw[0]}
  [337] = {x=20.02, y=-103, z=1, rx=-90, ry=68, fatherId=FrmDraw[0]}
  [338] = {x=19.94, y=-102.81, z=1, rx=-90, ry=68.05, fatherId=FrmDraw[0]}
  [339] = {x=19.87, y=-102.62, z=1, rx=-90, ry=68.09, fatherId=FrmDraw[0]}
  [340] = {x=19.79, y=-102.44, z=1, rx=-90, ry=68.13, fatherId=FrmDraw[0]}
  [341] = {x=19.72, y=-102.25, z=1, rx=-90, ry=68.17, fatherId=FrmDraw[0]}
  [342] = {x=19.64, y=-102.07, z=1, rx=-90, ry=68.21, fatherId=FrmDraw[0]}
  [343] = {x=19.57, y=-101.88, z=1, rx=-90, ry=68.25, fatherId=FrmDraw[0]}
  [344] = {x=19.49, y=-101.7, z=1, rx=-90, ry=68.3, fatherId=FrmDraw[0]}
  [345] = {x=19.42, y=-101.51, z=1, rx=-90, ry=68.34, fatherId=FrmDraw[0]}
  [346] = {x=19.35, y=-101.32, z=1, rx=-90, ry=68.38, fatherId=FrmDraw[0]}
  [347] = {x=19.27, y=-101.14, z=1, rx=-90, ry=68.42, fatherId=FrmDraw[0]}
  [348] = {x=19.2, y=-100.95, z=1, rx=-90, ry=68.46, fatherId=FrmDraw[0]}
  [349] = {x=19.13, y=-100.77, z=1, rx=-90, ry=68.5, fatherId=FrmDraw[0]}
  [350] = {x=19.05, y=-100.58, z=1, rx=-90, ry=68.55, fatherId=FrmDraw[0]}
  [351] = {x=18.98, y=-100.39, z=1, rx=-90, ry=68.59, fatherId=FrmDraw[0]}
  [352] = {x=18.91, y=-100.21, z=1, rx=-90, ry=68.63, fatherId=FrmDraw[0]}
  [353] = {x=18.83, y=-100.02, z=1, rx=-90, ry=68.67, fatherId=FrmDraw[0]}
  [354] = {x=18.76, y=-99.83, z=1, rx=-90, ry=68.71, fatherId=FrmDraw[0]}
  [355] = {x=18.69, y=-99.65, z=1, rx=-90, ry=68.75, fatherId=FrmDraw[0]}
  [356] = {x=18.62, y=-99.46, z=1, rx=-90, ry=68.8, fatherId=FrmDraw[0]}
  [357] = {x=18.54, y=-99.28, z=1, rx=-90, ry=68.84, fatherId=FrmDraw[0]}
  [358] = {x=18.47, y=-99.09, z=1, rx=-90, ry=68.88, fatherId=FrmDraw[0]}
  [359] = {x=18.4, y=-98.9, z=1, rx=-90, ry=68.92, fatherId=FrmDraw[0]}
  [360] = {x=18.33, y=-98.72, z=1, rx=-90, ry=68.96, fatherId=FrmDraw[0]}
  [361] = {x=18.26, y=-98.53, z=1, rx=-90, ry=69, fatherId=FrmDraw[0]}
  [362] = {x=18.19, y=-98.34, z=1, rx=-90, ry=69.05, fatherId=FrmDraw[0]}
  [363] = {x=18.11, y=-98.16, z=1, rx=-90, ry=69.09, fatherId=FrmDraw[0]}
  [364] = {x=18.04, y=-97.97, z=1, rx=-90, ry=69.13, fatherId=FrmDraw[0]}
  [365] = {x=17.97, y=-97.78, z=1, rx=-90, ry=69.17, fatherId=FrmDraw[0]}
  [366] = {x=17.9, y=-97.59, z=1, rx=-90, ry=69.21, fatherId=FrmDraw[0]}
  [367] = {x=17.83, y=-97.41, z=1, rx=-90, ry=69.25, fatherId=FrmDraw[0]}
  [368] = {x=17.76, y=-97.22, z=1, rx=-90, ry=69.3, fatherId=FrmDraw[0]}
  [369] = {x=17.69, y=-97.03, z=1, rx=-90, ry=69.34, fatherId=FrmDraw[0]}
  [370] = {x=17.62, y=-96.85, z=1, rx=-90, ry=69.38, fatherId=FrmDraw[0]}
  [371] = {x=17.55, y=-96.66, z=1, rx=-90, ry=69.42, fatherId=FrmDraw[0]}
  [372] = {x=17.48, y=-96.47, z=1, rx=-90, ry=69.46, fatherId=FrmDraw[0]}
  [373] = {x=17.41, y=-96.28, z=1, rx=-90, ry=69.5, fatherId=FrmDraw[0]}
  [374] = {x=17.34, y=-96.1, z=1, rx=-90, ry=69.55, fatherId=FrmDraw[0]}
  [375] = {x=17.27, y=-95.91, z=1, rx=-90, ry=69.59, fatherId=FrmDraw[0]}
  [376] = {x=17.2, y=-95.72, z=1, rx=-90, ry=69.63, fatherId=FrmDraw[0]}
  [377] = {x=17.13, y=-95.53, z=1, rx=-90, ry=69.67, fatherId=FrmDraw[0]}
  [378] = {x=17.06, y=-95.35, z=1, rx=-90, ry=69.71, fatherId=FrmDraw[0]}
  [379] = {x=16.99, y=-95.16, z=1, rx=-90, ry=69.75, fatherId=FrmDraw[0]}
  [380] = {x=16.92, y=-94.97, z=1, rx=-90, ry=69.8, fatherId=FrmDraw[0]}
  [381] = {x=16.85, y=-94.78, z=1, rx=-90, ry=69.84, fatherId=FrmDraw[0]}
  [382] = {x=16.78, y=-94.6, z=1, rx=-90, ry=69.88, fatherId=FrmDraw[0]}
  [383] = {x=16.71, y=-94.41, z=1, rx=-90, ry=69.92, fatherId=FrmDraw[0]}
  [384] = {x=16.64, y=-94.22, z=1, rx=-90, ry=69.96, fatherId=FrmDraw[0]}
  [385] = {x=16.58, y=-94.03, z=1, rx=-90, ry=70.01, fatherId=FrmDraw[0]}
  [386] = {x=16.51, y=-93.84, z=1, rx=-90, ry=70.05, fatherId=FrmDraw[0]}
  [387] = {x=16.44, y=-93.66, z=1, rx=-90, ry=70.09, fatherId=FrmDraw[0]}
  [388] = {x=16.37, y=-93.47, z=1, rx=-90, ry=70.13, fatherId=FrmDraw[0]}
  [389] = {x=16.3, y=-93.28, z=1, rx=-90, ry=70.17, fatherId=FrmDraw[0]}
  [390] = {x=16.24, y=-93.09, z=1, rx=-90, ry=70.21, fatherId=FrmDraw[0]}
  [391] = {x=16.17, y=-92.9, z=1, rx=-90, ry=70.26, fatherId=FrmDraw[0]}
  [392] = {x=16.1, y=-92.72, z=1, rx=-90, ry=70.3, fatherId=FrmDraw[0]}
  [393] = {x=16.03, y=-92.53, z=1, rx=-90, ry=70.34, fatherId=FrmDraw[0]}
  [394] = {x=15.97, y=-92.34, z=1, rx=-90, ry=70.38, fatherId=FrmDraw[0]}
  [395] = {x=15.9, y=-92.15, z=1, rx=-90, ry=70.42, fatherId=FrmDraw[0]}
  [396] = {x=15.83, y=-91.96, z=1, rx=-90, ry=70.46, fatherId=FrmDraw[0]}
  [397] = {x=15.77, y=-91.77, z=1, rx=-90, ry=70.5, fatherId=FrmDraw[0]}
  [398] = {x=15.7, y=-91.59, z=1, rx=-90, ry=70.55, fatherId=FrmDraw[0]}
  [399] = {x=15.63, y=-91.4, z=1, rx=-90, ry=70.59, fatherId=FrmDraw[0]}
  [400] = {x=15.57, y=-91.21, z=1, rx=-90, ry=70.63, fatherId=FrmDraw[0]}
  [401] = {x=15.5, y=-91.02, z=1, rx=-90, ry=70.67, fatherId=FrmDraw[0]}
  [402] = {x=15.43, y=-90.83, z=1, rx=-90, ry=70.71, fatherId=FrmDraw[0]}
  [403] = {x=15.37, y=-90.64, z=1, rx=-90, ry=70.76, fatherId=FrmDraw[0]}
  [404] = {x=15.3, y=-90.45, z=1, rx=-90, ry=70.8, fatherId=FrmDraw[0]}
  [405] = {x=15.24, y=-90.26, z=1, rx=-90, ry=70.84, fatherId=FrmDraw[0]}
  [406] = {x=15.17, y=-90.08, z=1, rx=-90, ry=70.88, fatherId=FrmDraw[0]}
  [407] = {x=15.1, y=-89.89, z=1, rx=-90, ry=70.92, fatherId=FrmDraw[0]}
  [408] = {x=15.04, y=-89.7, z=1, rx=-90, ry=70.96, fatherId=FrmDraw[0]}
  [409] = {x=14.97, y=-89.51, z=1, rx=-90, ry=71.01, fatherId=FrmDraw[0]}
  [410] = {x=14.91, y=-89.32, z=1, rx=-90, ry=71.05, fatherId=FrmDraw[0]}
  [411] = {x=14.84, y=-89.13, z=1, rx=-90, ry=71.09, fatherId=FrmDraw[0]}
  [412] = {x=14.78, y=-88.94, z=1, rx=-90, ry=71.13, fatherId=FrmDraw[0]}
  [413] = {x=14.72, y=-88.75, z=1, rx=-90, ry=71.17, fatherId=FrmDraw[0]}
  [414] = {x=14.65, y=-88.56, z=1, rx=-90, ry=71.21, fatherId=FrmDraw[0]}
  [415] = {x=14.59, y=-88.37, z=1, rx=-90, ry=71.26, fatherId=FrmDraw[0]}
  [416] = {x=14.52, y=-88.18, z=1, rx=-90, ry=71.3, fatherId=FrmDraw[0]}
  [417] = {x=14.46, y=-87.99, z=1, rx=-90, ry=71.34, fatherId=FrmDraw[0]}
  [418] = {x=14.39, y=-87.8, z=1, rx=-90, ry=71.38, fatherId=FrmDraw[0]}
  [419] = {x=14.33, y=-87.61, z=1, rx=-90, ry=71.42, fatherId=FrmDraw[0]}
  [420] = {x=14.27, y=-87.43, z=1, rx=-90, ry=71.46, fatherId=FrmDraw[0]}
  [421] = {x=14.2, y=-87.24, z=1, rx=-90, ry=71.51, fatherId=FrmDraw[0]}
  [422] = {x=14.14, y=-87.05, z=1, rx=-90, ry=71.55, fatherId=FrmDraw[0]}
  [423] = {x=14.08, y=-86.86, z=1, rx=-90, ry=71.59, fatherId=FrmDraw[0]}
  [424] = {x=14.01, y=-86.67, z=1, rx=-90, ry=71.63, fatherId=FrmDraw[0]}
  [425] = {x=13.95, y=-86.48, z=1, rx=-90, ry=71.67, fatherId=FrmDraw[0]}
  [426] = {x=13.89, y=-86.29, z=1, rx=-90, ry=71.71, fatherId=FrmDraw[0]}
  [427] = {x=13.82, y=-86.1, z=1, rx=-90, ry=71.76, fatherId=FrmDraw[0]}
  [428] = {x=13.76, y=-85.91, z=1, rx=-90, ry=71.8, fatherId=FrmDraw[0]}
  [429] = {x=13.7, y=-85.72, z=1, rx=-90, ry=71.84, fatherId=FrmDraw[0]}
  [430] = {x=13.64, y=-85.53, z=1, rx=-90, ry=71.88, fatherId=FrmDraw[0]}
  [431] = {x=13.58, y=-85.34, z=1, rx=-90, ry=71.92, fatherId=FrmDraw[0]}
  [432] = {x=13.51, y=-85.15, z=1, rx=-90, ry=71.96, fatherId=FrmDraw[0]}
  [433] = {x=13.45, y=-84.96, z=1, rx=-90, ry=72.01, fatherId=FrmDraw[0]}
  [434] = {x=13.39, y=-84.77, z=1, rx=-90, ry=72.05, fatherId=FrmDraw[0]}
  [435] = {x=13.33, y=-84.58, z=1, rx=-90, ry=72.09, fatherId=FrmDraw[0]}
  [436] = {x=13.27, y=-84.39, z=1, rx=-90, ry=72.13, fatherId=FrmDraw[0]}
  [437] = {x=13.21, y=-84.19, z=1, rx=-90, ry=72.17, fatherId=FrmDraw[0]}
  [438] = {x=13.14, y=-84, z=1, rx=-90, ry=72.21, fatherId=FrmDraw[0]}
  [439] = {x=13.08, y=-83.81, z=1, rx=-90, ry=72.26, fatherId=FrmDraw[0]}
  [440] = {x=13.02, y=-83.62, z=1, rx=-90, ry=72.3, fatherId=FrmDraw[0]}
  [441] = {x=12.96, y=-83.43, z=1, rx=-90, ry=72.34, fatherId=FrmDraw[0]}
  [442] = {x=12.9, y=-83.24, z=1, rx=-90, ry=72.38, fatherId=FrmDraw[0]}
  [443] = {x=12.84, y=-83.05, z=1, rx=-90, ry=72.42, fatherId=FrmDraw[0]}
  [444] = {x=12.78, y=-82.86, z=1, rx=-90, ry=72.46, fatherId=FrmDraw[0]}
  [445] = {x=12.72, y=-82.67, z=1, rx=-90, ry=72.51, fatherId=FrmDraw[0]}
  [446] = {x=12.66, y=-82.48, z=1, rx=-90, ry=72.55, fatherId=FrmDraw[0]}
  [447] = {x=12.6, y=-82.29, z=1, rx=-90, ry=72.59, fatherId=FrmDraw[0]}
  [448] = {x=12.54, y=-82.1, z=1, rx=-90, ry=72.63, fatherId=FrmDraw[0]}
  [449] = {x=12.48, y=-81.91, z=1, rx=-90, ry=72.67, fatherId=FrmDraw[0]}
  [450] = {x=12.42, y=-81.72, z=1, rx=-90, ry=72.71, fatherId=FrmDraw[0]}
  [451] = {x=12.36, y=-81.52, z=1, rx=-90, ry=72.76, fatherId=FrmDraw[0]}
  [452] = {x=12.3, y=-81.33, z=1, rx=-90, ry=72.8, fatherId=FrmDraw[0]}
  [453] = {x=12.24, y=-81.14, z=1, rx=-90, ry=72.84, fatherId=FrmDraw[0]}
  [454] = {x=12.18, y=-80.95, z=1, rx=-90, ry=72.88, fatherId=FrmDraw[0]}
  [455] = {x=12.13, y=-80.76, z=1, rx=-90, ry=72.92, fatherId=FrmDraw[0]}
  [456] = {x=12.07, y=-80.57, z=1, rx=-90, ry=72.96, fatherId=FrmDraw[0]}
  [457] = {x=12.01, y=-80.38, z=1, rx=-90, ry=73.01, fatherId=FrmDraw[0]}
  [458] = {x=11.95, y=-80.19, z=1, rx=-90, ry=73.05, fatherId=FrmDraw[0]}
  [459] = {x=11.89, y=-80, z=1, rx=-90, ry=73.09, fatherId=FrmDraw[0]}
  [460] = {x=11.83, y=-79.8, z=1, rx=-90, ry=73.13, fatherId=FrmDraw[0]}
  [461] = {x=11.78, y=-79.61, z=1, rx=-90, ry=73.17, fatherId=FrmDraw[0]}
  [462] = {x=11.72, y=-79.42, z=1, rx=-90, ry=73.21, fatherId=FrmDraw[0]}
  [463] = {x=11.66, y=-79.23, z=1, rx=-90, ry=73.26, fatherId=FrmDraw[0]}
  [464] = {x=11.6, y=-79.04, z=1, rx=-90, ry=73.3, fatherId=FrmDraw[0]}
  [465] = {x=11.55, y=-78.85, z=1, rx=-90, ry=73.34, fatherId=FrmDraw[0]}
  [466] = {x=11.49, y=-78.66, z=1, rx=-90, ry=73.38, fatherId=FrmDraw[0]}
  [467] = {x=11.43, y=-78.46, z=1, rx=-90, ry=73.42, fatherId=FrmDraw[0]}
  [468] = {x=11.37, y=-78.27, z=1, rx=-90, ry=73.46, fatherId=FrmDraw[0]}
  [469] = {x=11.32, y=-78.08, z=1, rx=-90, ry=73.51, fatherId=FrmDraw[0]}
  [470] = {x=11.26, y=-77.89, z=1, rx=-90, ry=73.55, fatherId=FrmDraw[0]}
  [471] = {x=11.2, y=-77.7, z=1, rx=-90, ry=73.59, fatherId=FrmDraw[0]}
  [472] = {x=11.15, y=-77.5, z=1, rx=-90, ry=73.63, fatherId=FrmDraw[0]}
  [473] = {x=11.09, y=-77.31, z=1, rx=-90, ry=73.67, fatherId=FrmDraw[0]}
  [474] = {x=11.04, y=-77.12, z=1, rx=-90, ry=73.71, fatherId=FrmDraw[0]}
  [475] = {x=10.98, y=-76.93, z=1, rx=-90, ry=73.76, fatherId=FrmDraw[0]}
  [476] = {x=10.92, y=-76.74, z=1, rx=-90, ry=73.8, fatherId=FrmDraw[0]}
  [477] = {x=10.87, y=-76.54, z=1, rx=-90, ry=73.84, fatherId=FrmDraw[0]}
  [478] = {x=10.81, y=-76.35, z=1, rx=-90, ry=73.88, fatherId=FrmDraw[0]}
  [479] = {x=10.76, y=-76.16, z=1, rx=-90, ry=73.92, fatherId=FrmDraw[0]}
  [480] = {x=10.7, y=-75.97, z=1, rx=-90, ry=73.96, fatherId=FrmDraw[0]}
  [481] = {x=10.65, y=-75.78, z=1, rx=-90, ry=74.01, fatherId=FrmDraw[0]}
  [482] = {x=10.59, y=-75.58, z=1, rx=-90, ry=74.05, fatherId=FrmDraw[0]}
  [483] = {x=10.54, y=-75.39, z=1, rx=-90, ry=74.09, fatherId=FrmDraw[0]}
  [484] = {x=10.48, y=-75.2, z=1, rx=-90, ry=74.13, fatherId=FrmDraw[0]}
  [485] = {x=10.43, y=-75.01, z=1, rx=-90, ry=74.17, fatherId=FrmDraw[0]}
  [486] = {x=10.37, y=-74.81, z=1, rx=-90, ry=74.21, fatherId=FrmDraw[0]}
  [487] = {x=10.32, y=-74.62, z=1, rx=-90, ry=74.26, fatherId=FrmDraw[0]}
  [488] = {x=10.26, y=-74.43, z=1, rx=-90, ry=74.3, fatherId=FrmDraw[0]}
  [489] = {x=10.21, y=-74.24, z=1, rx=-90, ry=74.34, fatherId=FrmDraw[0]}
  [490] = {x=10.16, y=-74.04, z=1, rx=-90, ry=74.38, fatherId=FrmDraw[0]}
  [491] = {x=10.1, y=-73.85, z=1, rx=-90, ry=74.42, fatherId=FrmDraw[0]}
  [492] = {x=10.05, y=-73.66, z=1, rx=-90, ry=74.46, fatherId=FrmDraw[0]}
  [493] = {x=9.99, y=-73.47, z=1, rx=-90, ry=74.51, fatherId=FrmDraw[0]}
  [494] = {x=9.94, y=-73.27, z=1, rx=-90, ry=74.55, fatherId=FrmDraw[0]}
  [495] = {x=9.89, y=-73.08, z=1, rx=-90, ry=74.59, fatherId=FrmDraw[0]}
  [496] = {x=9.84, y=-72.89, z=1, rx=-90, ry=74.63, fatherId=FrmDraw[0]}
  [497] = {x=9.78, y=-72.69, z=1, rx=-90, ry=74.67, fatherId=FrmDraw[0]}
  [498] = {x=9.73, y=-72.5, z=1, rx=-90, ry=74.71, fatherId=FrmDraw[0]}
  [499] = {x=9.68, y=-72.31, z=1, rx=-90, ry=74.76, fatherId=FrmDraw[0]}
  [500] = {x=9.62, y=-72.12, z=1, rx=-90, ry=74.8, fatherId=FrmDraw[0]}
  [501] = {x=9.57, y=-71.92, z=1, rx=-90, ry=74.84, fatherId=FrmDraw[0]}
  [502] = {x=9.52, y=-71.73, z=1, rx=-90, ry=74.88, fatherId=FrmDraw[0]}
  [503] = {x=9.47, y=-71.54, z=1, rx=-90, ry=74.92, fatherId=FrmDraw[0]}
  [504] = {x=9.42, y=-71.34, z=1, rx=-90, ry=74.96, fatherId=FrmDraw[0]}
  [505] = {x=9.36, y=-71.15, z=1, rx=-90, ry=75.01, fatherId=FrmDraw[0]}
  [506] = {x=9.31, y=-70.96, z=1, rx=-90, ry=75.05, fatherId=FrmDraw[0]}
  [507] = {x=9.26, y=-70.76, z=1, rx=-90, ry=75.09, fatherId=FrmDraw[0]}
  [508] = {x=9.21, y=-70.57, z=1, rx=-90, ry=75.13, fatherId=FrmDraw[0]}
  [509] = {x=9.16, y=-70.38, z=1, rx=-90, ry=75.17, fatherId=FrmDraw[0]}
  [510] = {x=9.11, y=-70.18, z=1, rx=-90, ry=75.21, fatherId=FrmDraw[0]}
  [511] = {x=9.06, y=-69.99, z=1, rx=-90, ry=75.26, fatherId=FrmDraw[0]}
  [512] = {x=9, y=-69.8, z=1, rx=-90, ry=75.3, fatherId=FrmDraw[0]}
  [513] = {x=8.95, y=-69.6, z=1, rx=-90, ry=75.34, fatherId=FrmDraw[0]}
  [514] = {x=8.9, y=-69.41, z=1, rx=-90, ry=75.38, fatherId=FrmDraw[0]}
  [515] = {x=8.85, y=-69.22, z=1, rx=-90, ry=75.42, fatherId=FrmDraw[0]}
  [516] = {x=8.8, y=-69.02, z=1, rx=-90, ry=75.46, fatherId=FrmDraw[0]}
  [517] = {x=8.75, y=-68.83, z=1, rx=-90, ry=75.51, fatherId=FrmDraw[0]}
  [518] = {x=8.7, y=-68.64, z=1, rx=-90, ry=75.55, fatherId=FrmDraw[0]}
  [519] = {x=8.65, y=-68.44, z=1, rx=-90, ry=75.59, fatherId=FrmDraw[0]}
  [520] = {x=8.6, y=-68.25, z=1, rx=-90, ry=75.63, fatherId=FrmDraw[0]}
  [521] = {x=8.55, y=-68.05, z=1, rx=-90, ry=75.67, fatherId=FrmDraw[0]}
  [522] = {x=8.5, y=-67.86, z=1, rx=-90, ry=75.71, fatherId=FrmDraw[0]}
  [523] = {x=8.46, y=-67.67, z=1, rx=-90, ry=75.76, fatherId=FrmDraw[0]}
  [524] = {x=8.41, y=-67.47, z=1, rx=-90, ry=75.8, fatherId=FrmDraw[0]}
  [525] = {x=8.36, y=-67.28, z=1, rx=-90, ry=75.84, fatherId=FrmDraw[0]}
  [526] = {x=8.31, y=-67.09, z=1, rx=-90, ry=75.88, fatherId=FrmDraw[0]}
  [527] = {x=8.26, y=-66.89, z=1, rx=-90, ry=75.92, fatherId=FrmDraw[0]}
  [528] = {x=8.21, y=-66.7, z=1, rx=-90, ry=75.96, fatherId=FrmDraw[0]}
  [529] = {x=8.16, y=-66.5, z=1, rx=-90, ry=76.01, fatherId=FrmDraw[0]}
  [530] = {x=8.11, y=-66.31, z=1, rx=-90, ry=76.05, fatherId=FrmDraw[0]}
  [531] = {x=8.07, y=-66.11, z=1, rx=-90, ry=76.09, fatherId=FrmDraw[0]}
  [532] = {x=8.02, y=-65.92, z=1, rx=-90, ry=76.13, fatherId=FrmDraw[0]}
  [533] = {x=7.97, y=-65.73, z=1, rx=-90, ry=76.17, fatherId=FrmDraw[0]}
  [534] = {x=7.92, y=-65.53, z=1, rx=-90, ry=76.21, fatherId=FrmDraw[0]}
  [535] = {x=7.87, y=-65.34, z=1, rx=-90, ry=76.26, fatherId=FrmDraw[0]}
  [536] = {x=7.83, y=-65.14, z=1, rx=-90, ry=76.3, fatherId=FrmDraw[0]}
  [537] = {x=7.78, y=-64.95, z=1, rx=-90, ry=76.34, fatherId=FrmDraw[0]}
  [538] = {x=7.73, y=-64.76, z=1, rx=-90, ry=76.38, fatherId=FrmDraw[0]}
  [539] = {x=7.69, y=-64.56, z=1, rx=-90, ry=76.42, fatherId=FrmDraw[0]}
  [540] = {x=7.64, y=-64.37, z=1, rx=-90, ry=76.46, fatherId=FrmDraw[0]}
  [541] = {x=7.59, y=-64.17, z=1, rx=-90, ry=76.51, fatherId=FrmDraw[0]}
  [542] = {x=7.55, y=-63.98, z=1, rx=-90, ry=76.55, fatherId=FrmDraw[0]}
  [543] = {x=7.5, y=-63.78, z=1, rx=-90, ry=76.59, fatherId=FrmDraw[0]}
  [544] = {x=7.45, y=-63.59, z=1, rx=-90, ry=76.63, fatherId=FrmDraw[0]}
  [545] = {x=7.41, y=-63.39, z=1, rx=-90, ry=76.67, fatherId=FrmDraw[0]}
  [546] = {x=7.36, y=-63.2, z=1, rx=-90, ry=76.71, fatherId=FrmDraw[0]}
  [547] = {x=7.31, y=-63, z=1, rx=-90, ry=76.76, fatherId=FrmDraw[0]}
  [548] = {x=7.27, y=-62.81, z=1, rx=-90, ry=76.8, fatherId=FrmDraw[0]}
  [549] = {x=7.22, y=-62.61, z=1, rx=-90, ry=76.84, fatherId=FrmDraw[0]}
  [550] = {x=7.18, y=-62.42, z=1, rx=-90, ry=76.88, fatherId=FrmDraw[0]}
  [551] = {x=7.13, y=-62.23, z=1, rx=-90, ry=76.92, fatherId=FrmDraw[0]}
  [552] = {x=7.09, y=-62.03, z=1, rx=-90, ry=76.96, fatherId=FrmDraw[0]}
  [553] = {x=7.04, y=-61.84, z=1, rx=-90, ry=77.01, fatherId=FrmDraw[0]}
  [554] = {x=7, y=-61.64, z=1, rx=-90, ry=77.05, fatherId=FrmDraw[0]}
  [555] = {x=6.95, y=-61.45, z=1, rx=-90, ry=77.09, fatherId=FrmDraw[0]}
  [556] = {x=6.91, y=-61.25, z=1, rx=-90, ry=77.13, fatherId=FrmDraw[0]}
  [557] = {x=6.86, y=-61.06, z=1, rx=-90, ry=77.17, fatherId=FrmDraw[0]}
  [558] = {x=6.82, y=-60.86, z=1, rx=-90, ry=77.21, fatherId=FrmDraw[0]}
  [559] = {x=6.77, y=-60.67, z=1, rx=-90, ry=77.26, fatherId=FrmDraw[0]}
  [560] = {x=6.73, y=-60.47, z=1, rx=-90, ry=77.3, fatherId=FrmDraw[0]}
  [561] = {x=6.69, y=-60.28, z=1, rx=-90, ry=77.34, fatherId=FrmDraw[0]}
  [562] = {x=6.64, y=-60.08, z=1, rx=-90, ry=77.38, fatherId=FrmDraw[0]}
  [563] = {x=6.6, y=-59.89, z=1, rx=-90, ry=77.42, fatherId=FrmDraw[0]}
  [564] = {x=6.56, y=-59.69, z=1, rx=-90, ry=77.46, fatherId=FrmDraw[0]}
  [565] = {x=6.51, y=-59.49, z=1, rx=-90, ry=77.51, fatherId=FrmDraw[0]}
  [566] = {x=6.47, y=-59.3, z=1, rx=-90, ry=77.55, fatherId=FrmDraw[0]}
  [567] = {x=6.43, y=-59.1, z=1, rx=-90, ry=77.59, fatherId=FrmDraw[0]}
  [568] = {x=6.38, y=-58.91, z=1, rx=-90, ry=77.63, fatherId=FrmDraw[0]}
  [569] = {x=6.34, y=-58.71, z=1, rx=-90, ry=77.67, fatherId=FrmDraw[0]}
  [570] = {x=6.3, y=-58.52, z=1, rx=-90, ry=77.71, fatherId=FrmDraw[0]}
  [571] = {x=6.26, y=-58.32, z=1, rx=-90, ry=77.76, fatherId=FrmDraw[0]}
  [572] = {x=6.21, y=-58.13, z=1, rx=-90, ry=77.8, fatherId=FrmDraw[0]}
  [573] = {x=6.17, y=-57.93, z=1, rx=-90, ry=77.84, fatherId=FrmDraw[0]}
  [574] = {x=6.13, y=-57.74, z=1, rx=-90, ry=77.88, fatherId=FrmDraw[0]}
  [575] = {x=6.09, y=-57.54, z=1, rx=-90, ry=77.92, fatherId=FrmDraw[0]}
  [576] = {x=6.05, y=-57.35, z=1, rx=-90, ry=77.96, fatherId=FrmDraw[0]}
  [577] = {x=6, y=-57.15, z=1, rx=-90, ry=78.01, fatherId=FrmDraw[0]}
  [578] = {x=5.96, y=-56.95, z=1, rx=-90, ry=78.05, fatherId=FrmDraw[0]}
  [579] = {x=5.92, y=-56.76, z=1, rx=-90, ry=78.09, fatherId=FrmDraw[0]}
  [580] = {x=5.88, y=-56.56, z=1, rx=-90, ry=78.13, fatherId=FrmDraw[0]}
  [581] = {x=5.84, y=-56.37, z=1, rx=-90, ry=78.17, fatherId=FrmDraw[0]}
  [582] = {x=5.8, y=-56.17, z=1, rx=-90, ry=78.21, fatherId=FrmDraw[0]}
  [583] = {x=5.76, y=-55.98, z=1, rx=-90, ry=78.26, fatherId=FrmDraw[0]}
  [584] = {x=5.72, y=-55.78, z=1, rx=-90, ry=78.3, fatherId=FrmDraw[0]}
  [585] = {x=5.68, y=-55.58, z=1, rx=-90, ry=78.34, fatherId=FrmDraw[0]}
  [586] = {x=5.64, y=-55.39, z=1, rx=-90, ry=78.38, fatherId=FrmDraw[0]}
  [587] = {x=5.6, y=-55.19, z=1, rx=-90, ry=78.42, fatherId=FrmDraw[0]}
  [588] = {x=5.56, y=-55, z=1, rx=-90, ry=78.46, fatherId=FrmDraw[0]}
  [589] = {x=5.52, y=-54.8, z=1, rx=-90, ry=78.51, fatherId=FrmDraw[0]}
  [590] = {x=5.48, y=-54.6, z=1, rx=-90, ry=78.55, fatherId=FrmDraw[0]}
  [591] = {x=5.44, y=-54.41, z=1, rx=-90, ry=78.59, fatherId=FrmDraw[0]}
  [592] = {x=5.4, y=-54.21, z=1, rx=-90, ry=78.63, fatherId=FrmDraw[0]}
  [593] = {x=5.36, y=-54.02, z=1, rx=-90, ry=78.67, fatherId=FrmDraw[0]}
  [594] = {x=5.32, y=-53.82, z=1, rx=-90, ry=78.71, fatherId=FrmDraw[0]}
  [595] = {x=5.28, y=-53.62, z=1, rx=-90, ry=78.76, fatherId=FrmDraw[0]}
  [596] = {x=5.24, y=-53.43, z=1, rx=-90, ry=78.8, fatherId=FrmDraw[0]}
  [597] = {x=5.2, y=-53.23, z=1, rx=-90, ry=78.84, fatherId=FrmDraw[0]}
  [598] = {x=5.16, y=-53.03, z=1, rx=-90, ry=78.88, fatherId=FrmDraw[0]}
  [599] = {x=5.12, y=-52.84, z=1, rx=-90, ry=78.92, fatherId=FrmDraw[0]}
  [600] = {x=5.09, y=-52.64, z=1, rx=-90, ry=78.96, fatherId=FrmDraw[0]}
  [601] = {x=5.05, y=-52.45, z=1, rx=-90, ry=79.01, fatherId=FrmDraw[0]}
  [602] = {x=5.01, y=-52.25, z=1, rx=-90, ry=79.05, fatherId=FrmDraw[0]}
  [603] = {x=4.97, y=-52.05, z=1, rx=-90, ry=79.09, fatherId=FrmDraw[0]}
  [604] = {x=4.93, y=-51.86, z=1, rx=-90, ry=79.13, fatherId=FrmDraw[0]}
  [605] = {x=4.9, y=-51.66, z=1, rx=-90, ry=79.17, fatherId=FrmDraw[0]}
  [606] = {x=4.86, y=-51.46, z=1, rx=-90, ry=79.21, fatherId=FrmDraw[0]}
  [607] = {x=4.82, y=-51.27, z=1, rx=-90, ry=79.26, fatherId=FrmDraw[0]}
  [608] = {x=4.78, y=-51.07, z=1, rx=-90, ry=79.3, fatherId=FrmDraw[0]}
  [609] = {x=4.75, y=-50.87, z=1, rx=-90, ry=79.34, fatherId=FrmDraw[0]}
  [610] = {x=4.71, y=-50.68, z=1, rx=-90, ry=79.38, fatherId=FrmDraw[0]}
  [611] = {x=4.67, y=-50.48, z=1, rx=-90, ry=79.42, fatherId=FrmDraw[0]}
  [612] = {x=4.64, y=-50.28, z=1, rx=-90, ry=79.46, fatherId=FrmDraw[0]}
  [613] = {x=4.6, y=-50.09, z=1, rx=-90, ry=79.51, fatherId=FrmDraw[0]}
  [614] = {x=4.56, y=-49.89, z=1, rx=-90, ry=79.55, fatherId=FrmDraw[0]}
  [615] = {x=4.53, y=-49.69, z=1, rx=-90, ry=79.59, fatherId=FrmDraw[0]}
  [616] = {x=4.49, y=-49.5, z=1, rx=-90, ry=79.63, fatherId=FrmDraw[0]}
  [617] = {x=4.46, y=-49.3, z=1, rx=-90, ry=79.67, fatherId=FrmDraw[0]}
  [618] = {x=4.42, y=-49.1, z=1, rx=-90, ry=79.71, fatherId=FrmDraw[0]}
  [619] = {x=4.38, y=-48.91, z=1, rx=-90, ry=79.76, fatherId=FrmDraw[0]}
  [620] = {x=4.35, y=-48.71, z=1, rx=-90, ry=79.8, fatherId=FrmDraw[0]}
  [621] = {x=4.31, y=-48.51, z=1, rx=-90, ry=79.84, fatherId=FrmDraw[0]}
  [622] = {x=4.28, y=-48.32, z=1, rx=-90, ry=79.88, fatherId=FrmDraw[0]}
  [623] = {x=4.24, y=-48.12, z=1, rx=-90, ry=79.92, fatherId=FrmDraw[0]}
  [624] = {x=4.21, y=-47.92, z=1, rx=-90, ry=79.96, fatherId=FrmDraw[0]}
  [625] = {x=4.17, y=-47.73, z=1, rx=-90, ry=80.01, fatherId=FrmDraw[0]}
  [626] = {x=4.14, y=-47.53, z=1, rx=-90, ry=80.05, fatherId=FrmDraw[0]}
  [627] = {x=4.1, y=-47.33, z=1, rx=-90, ry=80.09, fatherId=FrmDraw[0]}
  [628] = {x=4.07, y=-47.14, z=1, rx=-90, ry=80.13, fatherId=FrmDraw[0]}
  [629] = {x=4.04, y=-46.94, z=1, rx=-90, ry=80.17, fatherId=FrmDraw[0]}
  [630] = {x=4, y=-46.74, z=1, rx=-90, ry=80.21, fatherId=FrmDraw[0]}
  [631] = {x=3.97, y=-46.54, z=1, rx=-90, ry=80.26, fatherId=FrmDraw[0]}
  [632] = {x=3.93, y=-46.35, z=1, rx=-90, ry=80.3, fatherId=FrmDraw[0]}
  [633] = {x=3.9, y=-46.15, z=1, rx=-90, ry=80.34, fatherId=FrmDraw[0]}
  [634] = {x=3.87, y=-45.95, z=1, rx=-90, ry=80.38, fatherId=FrmDraw[0]}
  [635] = {x=3.83, y=-45.76, z=1, rx=-90, ry=80.42, fatherId=FrmDraw[0]}
  [636] = {x=3.8, y=-45.56, z=1, rx=-90, ry=80.46, fatherId=FrmDraw[0]}
  [637] = {x=3.77, y=-45.36, z=1, rx=-90, ry=80.51, fatherId=FrmDraw[0]}
  [638] = {x=3.73, y=-45.16, z=1, rx=-90, ry=80.55, fatherId=FrmDraw[0]}
  [639] = {x=3.7, y=-44.97, z=1, rx=-90, ry=80.59, fatherId=FrmDraw[0]}
  [640] = {x=3.67, y=-44.77, z=1, rx=-90, ry=80.63, fatherId=FrmDraw[0]}
  [641] = {x=3.64, y=-44.57, z=1, rx=-90, ry=80.67, fatherId=FrmDraw[0]}
  [642] = {x=3.6, y=-44.37, z=1, rx=-90, ry=80.71, fatherId=FrmDraw[0]}
  [643] = {x=3.57, y=-44.18, z=1, rx=-90, ry=80.76, fatherId=FrmDraw[0]}
  [644] = {x=3.54, y=-43.98, z=1, rx=-90, ry=80.8, fatherId=FrmDraw[0]}
  [645] = {x=3.51, y=-43.78, z=1, rx=-90, ry=80.84, fatherId=FrmDraw[0]}
  [646] = {x=3.48, y=-43.58, z=1, rx=-90, ry=80.88, fatherId=FrmDraw[0]}
  [647] = {x=3.44, y=-43.39, z=1, rx=-90, ry=80.92, fatherId=FrmDraw[0]}
  [648] = {x=3.41, y=-43.19, z=1, rx=-90, ry=80.96, fatherId=FrmDraw[0]}
  [649] = {x=3.38, y=-42.99, z=1, rx=-90, ry=81.01, fatherId=FrmDraw[0]}
  [650] = {x=3.35, y=-42.79, z=1, rx=-90, ry=81.05, fatherId=FrmDraw[0]}
  [651] = {x=3.32, y=-42.6, z=1, rx=-90, ry=81.09, fatherId=FrmDraw[0]}
  [652] = {x=3.29, y=-42.4, z=1, rx=-90, ry=81.13, fatherId=FrmDraw[0]}
  [653] = {x=3.26, y=-42.2, z=1, rx=-90, ry=81.17, fatherId=FrmDraw[0]}
  [654] = {x=3.23, y=-42, z=1, rx=-90, ry=81.21, fatherId=FrmDraw[0]}
  [655] = {x=3.2, y=-41.81, z=1, rx=-90, ry=81.26, fatherId=FrmDraw[0]}
  [656] = {x=3.17, y=-41.61, z=1, rx=-90, ry=81.3, fatherId=FrmDraw[0]}
  [657] = {x=3.14, y=-41.41, z=1, rx=-90, ry=81.34, fatherId=FrmDraw[0]}
  [658] = {x=3.11, y=-41.21, z=1, rx=-90, ry=81.38, fatherId=FrmDraw[0]}
  [659] = {x=3.08, y=-41.02, z=1, rx=-90, ry=81.42, fatherId=FrmDraw[0]}
  [660] = {x=3.05, y=-40.82, z=1, rx=-90, ry=81.46, fatherId=FrmDraw[0]}
  [661] = {x=3.02, y=-40.62, z=1, rx=-90, ry=81.51, fatherId=FrmDraw[0]}
  [662] = {x=2.99, y=-40.42, z=1, rx=-90, ry=81.55, fatherId=FrmDraw[0]}
  [663] = {x=2.96, y=-40.22, z=1, rx=-90, ry=81.59, fatherId=FrmDraw[0]}
  [664] = {x=2.93, y=-40.03, z=1, rx=-90, ry=81.63, fatherId=FrmDraw[0]}
  [665] = {x=2.9, y=-39.83, z=1, rx=-90, ry=81.67, fatherId=FrmDraw[0]}
  [666] = {x=2.87, y=-39.63, z=1, rx=-90, ry=81.71, fatherId=FrmDraw[0]}
  [667] = {x=2.84, y=-39.43, z=1, rx=-90, ry=81.76, fatherId=FrmDraw[0]}
  [668] = {x=2.81, y=-39.23, z=1, rx=-90, ry=81.8, fatherId=FrmDraw[0]}
  [669] = {x=2.78, y=-39.04, z=1, rx=-90, ry=81.84, fatherId=FrmDraw[0]}
  [670] = {x=2.76, y=-38.84, z=1, rx=-90, ry=81.88, fatherId=FrmDraw[0]}
  [671] = {x=2.73, y=-38.64, z=1, rx=-90, ry=81.92, fatherId=FrmDraw[0]}
  [672] = {x=2.7, y=-38.44, z=1, rx=-90, ry=81.96, fatherId=FrmDraw[0]}
  [673] = {x=2.67, y=-38.24, z=1, rx=-90, ry=82.01, fatherId=FrmDraw[0]}
  [674] = {x=2.64, y=-38.05, z=1, rx=-90, ry=82.05, fatherId=FrmDraw[0]}
  [675] = {x=2.62, y=-37.85, z=1, rx=-90, ry=82.09, fatherId=FrmDraw[0]}
  [676] = {x=2.59, y=-37.65, z=1, rx=-90, ry=82.13, fatherId=FrmDraw[0]}
  [677] = {x=2.56, y=-37.45, z=1, rx=-90, ry=82.17, fatherId=FrmDraw[0]}
  [678] = {x=2.54, y=-37.25, z=1, rx=-90, ry=82.21, fatherId=FrmDraw[0]}
  [679] = {x=2.51, y=-37.06, z=1, rx=-90, ry=82.26, fatherId=FrmDraw[0]}
  [680] = {x=2.48, y=-36.86, z=1, rx=-90, ry=82.3, fatherId=FrmDraw[0]}
  [681] = {x=2.45, y=-36.66, z=1, rx=-90, ry=82.34, fatherId=FrmDraw[0]}
  [682] = {x=2.43, y=-36.46, z=1, rx=-90, ry=82.38, fatherId=FrmDraw[0]}
  [683] = {x=2.4, y=-36.26, z=1, rx=-90, ry=82.42, fatherId=FrmDraw[0]}
  [684] = {x=2.38, y=-36.06, z=1, rx=-90, ry=82.46, fatherId=FrmDraw[0]}
  [685] = {x=2.35, y=-35.87, z=1, rx=-90, ry=82.51, fatherId=FrmDraw[0]}
  [686] = {x=2.32, y=-35.67, z=1, rx=-90, ry=82.55, fatherId=FrmDraw[0]}
  [687] = {x=2.3, y=-35.47, z=1, rx=-90, ry=82.59, fatherId=FrmDraw[0]}
  [688] = {x=2.27, y=-35.27, z=1, rx=-90, ry=82.63, fatherId=FrmDraw[0]}
  [689] = {x=2.25, y=-35.07, z=1, rx=-90, ry=82.67, fatherId=FrmDraw[0]}
  [690] = {x=2.22, y=-34.87, z=1, rx=-90, ry=82.71, fatherId=FrmDraw[0]}
  [691] = {x=2.2, y=-34.68, z=1, rx=-90, ry=82.76, fatherId=FrmDraw[0]}
  [692] = {x=2.17, y=-34.48, z=1, rx=-90, ry=82.8, fatherId=FrmDraw[0]}
  [693] = {x=2.14, y=-34.28, z=1, rx=-90, ry=82.84, fatherId=FrmDraw[0]}
  [694] = {x=2.12, y=-34.08, z=1, rx=-90, ry=82.88, fatherId=FrmDraw[0]}
  [695] = {x=2.1, y=-33.88, z=1, rx=-90, ry=82.92, fatherId=FrmDraw[0]}
  [696] = {x=2.07, y=-33.68, z=1, rx=-90, ry=82.96, fatherId=FrmDraw[0]}
  [697] = {x=2.05, y=-33.49, z=1, rx=-90, ry=83.01, fatherId=FrmDraw[0]}
  [698] = {x=2.02, y=-33.29, z=1, rx=-90, ry=83.05, fatherId=FrmDraw[0]}
  [699] = {x=2, y=-33.09, z=1, rx=-90, ry=83.09, fatherId=FrmDraw[0]}
  [700] = {x=1.97, y=-32.89, z=1, rx=-90, ry=83.13, fatherId=FrmDraw[0]}
  [701] = {x=1.95, y=-32.69, z=1, rx=-90, ry=83.17, fatherId=FrmDraw[0]}
  [702] = {x=1.93, y=-32.49, z=1, rx=-90, ry=83.21, fatherId=FrmDraw[0]}
  [703] = {x=1.9, y=-32.29, z=1, rx=-90, ry=83.26, fatherId=FrmDraw[0]}
  [704] = {x=1.88, y=-32.1, z=1, rx=-90, ry=83.3, fatherId=FrmDraw[0]}
  [705] = {x=1.86, y=-31.9, z=1, rx=-90, ry=83.34, fatherId=FrmDraw[0]}
  [706] = {x=1.83, y=-31.7, z=1, rx=-90, ry=83.38, fatherId=FrmDraw[0]}
  [707] = {x=1.81, y=-31.5, z=1, rx=-90, ry=83.42, fatherId=FrmDraw[0]}
  [708] = {x=1.79, y=-31.3, z=1, rx=-90, ry=83.46, fatherId=FrmDraw[0]}
  [709] = {x=1.76, y=-31.1, z=1, rx=-90, ry=83.51, fatherId=FrmDraw[0]}
  [710] = {x=1.74, y=-30.9, z=1, rx=-90, ry=83.55, fatherId=FrmDraw[0]}
  [711] = {x=1.72, y=-30.7, z=1, rx=-90, ry=83.59, fatherId=FrmDraw[0]}
  [712] = {x=1.7, y=-30.51, z=1, rx=-90, ry=83.63, fatherId=FrmDraw[0]}
  [713] = {x=1.68, y=-30.31, z=1, rx=-90, ry=83.67, fatherId=FrmDraw[0]}
  [714] = {x=1.65, y=-30.11, z=1, rx=-90, ry=83.71, fatherId=FrmDraw[0]}
  [715] = {x=1.63, y=-29.91, z=1, rx=-90, ry=83.76, fatherId=FrmDraw[0]}
  [716] = {x=1.61, y=-29.71, z=1, rx=-90, ry=83.8, fatherId=FrmDraw[0]}
  [717] = {x=1.59, y=-29.51, z=1, rx=-90, ry=83.84, fatherId=FrmDraw[0]}
  [718] = {x=1.57, y=-29.31, z=1, rx=-90, ry=83.88, fatherId=FrmDraw[0]}
  [719] = {x=1.55, y=-29.11, z=1, rx=-90, ry=83.92, fatherId=FrmDraw[0]}
  [720] = {x=1.52, y=-28.92, z=1, rx=-90, ry=83.96, fatherId=FrmDraw[0]}
  [721] = {x=1.5, y=-28.72, z=1, rx=-90, ry=84.01, fatherId=FrmDraw[0]}
  [722] = {x=1.48, y=-28.52, z=1, rx=-90, ry=84.05, fatherId=FrmDraw[0]}
  [723] = {x=1.46, y=-28.32, z=1, rx=-90, ry=84.09, fatherId=FrmDraw[0]}
  [724] = {x=1.44, y=-28.12, z=1, rx=-90, ry=84.13, fatherId=FrmDraw[0]}
  [725] = {x=1.42, y=-27.92, z=1, rx=-90, ry=84.17, fatherId=FrmDraw[0]}
  [726] = {x=1.4, y=-27.72, z=1, rx=-90, ry=84.21, fatherId=FrmDraw[0]}
  [727] = {x=1.38, y=-27.52, z=1, rx=-90, ry=84.26, fatherId=FrmDraw[0]}
  [728] = {x=1.36, y=-27.32, z=1, rx=-90, ry=84.3, fatherId=FrmDraw[0]}
  [729] = {x=1.34, y=-27.12, z=1, rx=-90, ry=84.34, fatherId=FrmDraw[0]}
  [730] = {x=1.32, y=-26.93, z=1, rx=-90, ry=84.38, fatherId=FrmDraw[0]}
  [731] = {x=1.3, y=-26.73, z=1, rx=-90, ry=84.42, fatherId=FrmDraw[0]}
  [732] = {x=1.28, y=-26.53, z=1, rx=-90, ry=84.46, fatherId=FrmDraw[0]}
  [733] = {x=1.26, y=-26.33, z=1, rx=-90, ry=84.51, fatherId=FrmDraw[0]}
  [734] = {x=1.24, y=-26.13, z=1, rx=-90, ry=84.55, fatherId=FrmDraw[0]}
  [735] = {x=1.23, y=-25.93, z=1, rx=-90, ry=84.59, fatherId=FrmDraw[0]}
  [736] = {x=1.21, y=-25.73, z=1, rx=-90, ry=84.63, fatherId=FrmDraw[0]}
  [737] = {x=1.19, y=-25.53, z=1, rx=-90, ry=84.67, fatherId=FrmDraw[0]}
  [738] = {x=1.17, y=-25.33, z=1, rx=-90, ry=84.71, fatherId=FrmDraw[0]}
  [739] = {x=1.15, y=-25.13, z=1, rx=-90, ry=84.76, fatherId=FrmDraw[0]}
  [740] = {x=1.13, y=-24.93, z=1, rx=-90, ry=84.8, fatherId=FrmDraw[0]}
  [741] = {x=1.11, y=-24.74, z=1, rx=-90, ry=84.84, fatherId=FrmDraw[0]}
  [742] = {x=1.1, y=-24.54, z=1, rx=-90, ry=84.88, fatherId=FrmDraw[0]}
  [743] = {x=1.08, y=-24.34, z=1, rx=-90, ry=84.92, fatherId=FrmDraw[0]}
  [744] = {x=1.06, y=-24.14, z=1, rx=-90, ry=84.96, fatherId=FrmDraw[0]}
  [745] = {x=1.04, y=-23.94, z=1, rx=-90, ry=85.01, fatherId=FrmDraw[0]}
  [746] = {x=1.03, y=-23.74, z=1, rx=-90, ry=85.05, fatherId=FrmDraw[0]}
  [747] = {x=1.01, y=-23.54, z=1, rx=-90, ry=85.09, fatherId=FrmDraw[0]}
  [748] = {x=0.99, y=-23.34, z=1, rx=-90, ry=85.13, fatherId=FrmDraw[0]}
  [749] = {x=0.98, y=-23.14, z=1, rx=-90, ry=85.17, fatherId=FrmDraw[0]}
  [750] = {x=0.96, y=-22.94, z=1, rx=-90, ry=85.21, fatherId=FrmDraw[0]}
  [751] = {x=0.94, y=-22.74, z=1, rx=-90, ry=85.26, fatherId=FrmDraw[0]}
  [752] = {x=0.93, y=-22.54, z=1, rx=-90, ry=85.3, fatherId=FrmDraw[0]}
  [753] = {x=0.91, y=-22.34, z=1, rx=-90, ry=85.34, fatherId=FrmDraw[0]}
  [754] = {x=0.89, y=-22.14, z=1, rx=-90, ry=85.38, fatherId=FrmDraw[0]}
  [755] = {x=0.88, y=-21.95, z=1, rx=-90, ry=85.42, fatherId=FrmDraw[0]}
  [756] = {x=0.86, y=-21.75, z=1, rx=-90, ry=85.46, fatherId=FrmDraw[0]}
  [757] = {x=0.85, y=-21.55, z=1, rx=-90, ry=85.51, fatherId=FrmDraw[0]}
  [758] = {x=0.83, y=-21.35, z=1, rx=-90, ry=85.55, fatherId=FrmDraw[0]}
  [759] = {x=0.81, y=-21.15, z=1, rx=-90, ry=85.59, fatherId=FrmDraw[0]}
  [760] = {x=0.8, y=-20.95, z=1, rx=-90, ry=85.63, fatherId=FrmDraw[0]}
  [761] = {x=0.78, y=-20.75, z=1, rx=-90, ry=85.67, fatherId=FrmDraw[0]}
  [762] = {x=0.77, y=-20.55, z=1, rx=-90, ry=85.71, fatherId=FrmDraw[0]}
  [763] = {x=0.75, y=-20.35, z=1, rx=-90, ry=85.76, fatherId=FrmDraw[0]}
  [764] = {x=0.74, y=-20.15, z=1, rx=-90, ry=85.8, fatherId=FrmDraw[0]}
  [765] = {x=0.72, y=-19.95, z=1, rx=-90, ry=85.84, fatherId=FrmDraw[0]}
  [766] = {x=0.71, y=-19.75, z=1, rx=-90, ry=85.88, fatherId=FrmDraw[0]}
  [767] = {x=0.7, y=-19.55, z=1, rx=-90, ry=85.92, fatherId=FrmDraw[0]}
  [768] = {x=0.68, y=-19.35, z=1, rx=-90, ry=85.96, fatherId=FrmDraw[0]}
  [769] = {x=0.67, y=-19.15, z=1, rx=-90, ry=86.01, fatherId=FrmDraw[0]}
  [770] = {x=0.65, y=-18.95, z=1, rx=-90, ry=86.05, fatherId=FrmDraw[0]}
  [771] = {x=0.64, y=-18.75, z=1, rx=-90, ry=86.09, fatherId=FrmDraw[0]}
  [772] = {x=0.63, y=-18.55, z=1, rx=-90, ry=86.13, fatherId=FrmDraw[0]}
  [773] = {x=0.61, y=-18.36, z=1, rx=-90, ry=86.17, fatherId=FrmDraw[0]}
  [774] = {x=0.6, y=-18.16, z=1, rx=-90, ry=86.21, fatherId=FrmDraw[0]}
  [775] = {x=0.59, y=-17.96, z=1, rx=-90, ry=86.26, fatherId=FrmDraw[0]}
  [776] = {x=0.57, y=-17.76, z=1, rx=-90, ry=86.3, fatherId=FrmDraw[0]}
  [777] = {x=0.56, y=-17.56, z=1, rx=-90, ry=86.34, fatherId=FrmDraw[0]}
  [778] = {x=0.55, y=-17.36, z=1, rx=-90, ry=86.38, fatherId=FrmDraw[0]}
  [779] = {x=0.54, y=-17.16, z=1, rx=-90, ry=86.42, fatherId=FrmDraw[0]}
  [780] = {x=0.52, y=-16.96, z=1, rx=-90, ry=86.46, fatherId=FrmDraw[0]}
  [781] = {x=0.51, y=-16.76, z=1, rx=-90, ry=86.51, fatherId=FrmDraw[0]}
  [782] = {x=0.5, y=-16.56, z=1, rx=-90, ry=86.55, fatherId=FrmDraw[0]}
  [783] = {x=0.49, y=-16.36, z=1, rx=-90, ry=86.59, fatherId=FrmDraw[0]}
  [784] = {x=0.48, y=-16.16, z=1, rx=-90, ry=86.63, fatherId=FrmDraw[0]}
  [785] = {x=0.46, y=-15.96, z=1, rx=-90, ry=86.67, fatherId=FrmDraw[0]}
  [786] = {x=0.45, y=-15.76, z=1, rx=-90, ry=86.71, fatherId=FrmDraw[0]}
  [787] = {x=0.44, y=-15.56, z=1, rx=-90, ry=86.76, fatherId=FrmDraw[0]}
  [788] = {x=0.43, y=-15.36, z=1, rx=-90, ry=86.8, fatherId=FrmDraw[0]}
  [789] = {x=0.42, y=-15.16, z=1, rx=-90, ry=86.84, fatherId=FrmDraw[0]}
  [790] = {x=0.41, y=-14.96, z=1, rx=-90, ry=86.88, fatherId=FrmDraw[0]}
  [791] = {x=0.4, y=-14.76, z=1, rx=-90, ry=86.92, fatherId=FrmDraw[0]}
  [792] = {x=0.39, y=-14.56, z=1, rx=-90, ry=86.96, fatherId=FrmDraw[0]}
  [793] = {x=0.38, y=-14.36, z=1, rx=-90, ry=87.01, fatherId=FrmDraw[0]}
  [794] = {x=0.36, y=-14.16, z=1, rx=-90, ry=87.05, fatherId=FrmDraw[0]}
  [795] = {x=0.35, y=-13.96, z=1, rx=-90, ry=87.09, fatherId=FrmDraw[0]}
  [796] = {x=0.34, y=-13.76, z=1, rx=-90, ry=87.13, fatherId=FrmDraw[0]}
  [797] = {x=0.33, y=-13.56, z=1, rx=-90, ry=87.17, fatherId=FrmDraw[0]}
  [798] = {x=0.32, y=-13.36, z=1, rx=-90, ry=87.21, fatherId=FrmDraw[0]}
  [799] = {x=0.32, y=-13.16, z=1, rx=-90, ry=87.26, fatherId=FrmDraw[0]}
  [800] = {x=0.31, y=-12.96, z=1, rx=-90, ry=87.3, fatherId=FrmDraw[0]}
  [801] = {x=0.3, y=-12.76, z=1, rx=-90, ry=87.34, fatherId=FrmDraw[0]}
  [802] = {x=0.29, y=-12.56, z=1, rx=-90, ry=87.38, fatherId=FrmDraw[0]}
  [803] = {x=0.28, y=-12.36, z=1, rx=-90, ry=87.42, fatherId=FrmDraw[0]}
  [804] = {x=0.27, y=-12.17, z=1, rx=-90, ry=87.46, fatherId=FrmDraw[0]}
  [805] = {x=0.26, y=-11.97, z=1, rx=-90, ry=87.51, fatherId=FrmDraw[0]}
  [806] = {x=0.25, y=-11.77, z=1, rx=-90, ry=87.55, fatherId=FrmDraw[0]}
  [807] = {x=0.24, y=-11.57, z=1, rx=-90, ry=87.59, fatherId=FrmDraw[0]}
  [808] = {x=0.23, y=-11.37, z=1, rx=-90, ry=87.63, fatherId=FrmDraw[0]}
  [809] = {x=0.23, y=-11.17, z=1, rx=-90, ry=87.67, fatherId=FrmDraw[0]}
  [810] = {x=0.22, y=-10.97, z=1, rx=-90, ry=87.71, fatherId=FrmDraw[0]}
  [811] = {x=0.21, y=-10.77, z=1, rx=-90, ry=87.76, fatherId=FrmDraw[0]}
  [812] = {x=0.2, y=-10.57, z=1, rx=-90, ry=87.8, fatherId=FrmDraw[0]}
  [813] = {x=0.2, y=-10.37, z=1, rx=-90, ry=87.84, fatherId=FrmDraw[0]}
  [814] = {x=0.19, y=-10.17, z=1, rx=-90, ry=87.88, fatherId=FrmDraw[0]}
  [815] = {x=0.18, y=-9.97, z=1, rx=-90, ry=87.92, fatherId=FrmDraw[0]}
  [816] = {x=0.17, y=-9.77, z=1, rx=-90, ry=87.96, fatherId=FrmDraw[0]}
  [817] = {x=0.17, y=-9.57, z=1, rx=-90, ry=88.01, fatherId=FrmDraw[0]}
  [818] = {x=0.16, y=-9.37, z=1, rx=-90, ry=88.05, fatherId=FrmDraw[0]}
  [819] = {x=0.15, y=-9.17, z=1, rx=-90, ry=88.09, fatherId=FrmDraw[0]}
  [820] = {x=0.15, y=-8.97, z=1, rx=-90, ry=88.13, fatherId=FrmDraw[0]}
  [821] = {x=0.14, y=-8.77, z=1, rx=-90, ry=88.17, fatherId=FrmDraw[0]}
  [822] = {x=0.13, y=-8.57, z=1, rx=-90, ry=88.21, fatherId=FrmDraw[0]}
  [823] = {x=0.13, y=-8.37, z=1, rx=-90, ry=88.26, fatherId=FrmDraw[0]}
  [824] = {x=0.12, y=-8.17, z=1, rx=-90, ry=88.3, fatherId=FrmDraw[0]}
  [825] = {x=0.12, y=-7.97, z=1, rx=-90, ry=88.34, fatherId=FrmDraw[0]}
  [826] = {x=0.11, y=-7.77, z=1, rx=-90, ry=88.38, fatherId=FrmDraw[0]}
  [827] = {x=0.1, y=-7.57, z=1, rx=-90, ry=88.42, fatherId=FrmDraw[0]}
  [828] = {x=0.1, y=-7.37, z=1, rx=-90, ry=88.46, fatherId=FrmDraw[0]}
  [829] = {x=0.09, y=-7.17, z=1, rx=-90, ry=88.51, fatherId=FrmDraw[0]}
  [830] = {x=0.09, y=-6.97, z=1, rx=-90, ry=88.55, fatherId=FrmDraw[0]}
  [831] = {x=0.08, y=-6.77, z=1, rx=-90, ry=88.59, fatherId=FrmDraw[0]}
  [832] = {x=0.08, y=-6.57, z=1, rx=-90, ry=88.63, fatherId=FrmDraw[0]}
  [833] = {x=0.07, y=-6.37, z=1, rx=-90, ry=88.67, fatherId=FrmDraw[0]}
  [834] = {x=0.07, y=-6.17, z=1, rx=-90, ry=88.71, fatherId=FrmDraw[0]}
  [835] = {x=0.06, y=-5.97, z=1, rx=-90, ry=88.76, fatherId=FrmDraw[0]}
  [836] = {x=0.06, y=-5.77, z=1, rx=-90, ry=88.8, fatherId=FrmDraw[0]}
  [837] = {x=0.06, y=-5.57, z=1, rx=-90, ry=88.84, fatherId=FrmDraw[0]}
  [838] = {x=0.05, y=-5.37, z=1, rx=-90, ry=88.88, fatherId=FrmDraw[0]}
  [839] = {x=0.05, y=-5.17, z=1, rx=-90, ry=88.92, fatherId=FrmDraw[0]}
  [840] = {x=0.04, y=-4.97, z=1, rx=-90, ry=88.96, fatherId=FrmDraw[0]}
  [841] = {x=0.04, y=-4.77, z=1, rx=-90, ry=89.01, fatherId=FrmDraw[0]}
  [842] = {x=0.04, y=-4.57, z=1, rx=-90, ry=89.05, fatherId=FrmDraw[0]}
  [843] = {x=0.03, y=-4.37, z=1, rx=-90, ry=89.09, fatherId=FrmDraw[0]}
  [844] = {x=0.03, y=-4.17, z=1, rx=-90, ry=89.13, fatherId=FrmDraw[0]}
  [845] = {x=0.03, y=-3.97, z=1, rx=-90, ry=89.17, fatherId=FrmDraw[0]}
  [846] = {x=0.03, y=-3.77, z=1, rx=-90, ry=89.21, fatherId=FrmDraw[0]}
  [847] = {x=0.02, y=-3.57, z=1, rx=-90, ry=89.26, fatherId=FrmDraw[0]}
  [848] = {x=0.02, y=-3.37, z=1, rx=-90, ry=89.3, fatherId=FrmDraw[0]}
  [849] = {x=0.02, y=-3.17, z=1, rx=-90, ry=89.34, fatherId=FrmDraw[0]}
  [850] = {x=0.02, y=-2.97, z=1, rx=-90, ry=89.38, fatherId=FrmDraw[0]}
  [851] = {x=0.01, y=-2.77, z=1, rx=-90, ry=89.42, fatherId=FrmDraw[0]}
  [852] = {x=0.01, y=-2.57, z=1, rx=-90, ry=89.46, fatherId=FrmDraw[0]}
  [853] = {x=0.01, y=-2.37, z=1, rx=-90, ry=89.51, fatherId=FrmDraw[0]}
  [854] = {x=0.01, y=-2.17, z=1, rx=-90, ry=89.55, fatherId=FrmDraw[0]}
  [855] = {x=0.01, y=-1.97, z=1, rx=-90, ry=89.59, fatherId=FrmDraw[0]}
  [856] = {x=0.01, y=-1.77, z=1, rx=-90, ry=89.63, fatherId=FrmDraw[0]}
  [857] = {y=-1.57, z=1, rx=-90, ry=89.67, fatherId=FrmDraw[0]}
  [858] = {y=-1.37, z=1, rx=-90, ry=89.71, fatherId=FrmDraw[0]}
  [859] = {y=-1.17, z=1, rx=-90, ry=89.76, fatherId=FrmDraw[0]}
  [860] = {y=-0.97, z=1, rx=-90, ry=89.8, fatherId=FrmDraw[0]}
  [861] = {y=-0.77, z=1, rx=-90, ry=89.84, fatherId=FrmDraw[0]}
  [862] = {y=-0.57, z=1, rx=-90, ry=89.88, fatherId=FrmDraw[0]}
  [863] = {y=-0.37, z=1, rx=-90, ry=89.92, fatherId=FrmDraw[0]}
  [864] = {y=-0.17, z=1, rx=-90, ry=89.96, fatherId=FrmDraw[0]}
  [865] = {y=0.03, z=1, rx=90, ry=89.99, fatherId=FrmDraw[0]}
  [866] = {y=0.23, z=1, rx=90, ry=89.95, fatherId=FrmDraw[0]}
  [867] = {y=0.43, z=1, rx=90, ry=89.91, fatherId=FrmDraw[0]}
  [868] = {y=0.63, z=1, rx=90, ry=89.87, fatherId=FrmDraw[0]}
  [869] = {y=0.83, z=1, rx=90, ry=89.83, fatherId=FrmDraw[0]}
  [870] = {y=1.03, z=1, rx=90, ry=89.79, fatherId=FrmDraw[0]}
  [871] = {y=1.23, z=1, rx=90, ry=89.74, fatherId=FrmDraw[0]}
  [872] = {y=1.43, z=1, rx=90, ry=89.7, fatherId=FrmDraw[0]}
  [873] = {y=1.63, z=1, rx=90, ry=89.66, fatherId=FrmDraw[0]}
  [874] = {x=0.01, y=1.83, z=1, rx=90, ry=89.62, fatherId=FrmDraw[0]}
  [875] = {x=0.01, y=2.03, z=1, rx=90, ry=89.58, fatherId=FrmDraw[0]}
  [876] = {x=0.01, y=2.23, z=1, rx=90, ry=89.54, fatherId=FrmDraw[0]}
  [877] = {x=0.01, y=2.43, z=1, rx=90, ry=89.49, fatherId=FrmDraw[0]}
  [878] = {x=0.01, y=2.63, z=1, rx=90, ry=89.45, fatherId=FrmDraw[0]}
  [879] = {x=0.01, y=2.83, z=1, rx=90, ry=89.41, fatherId=FrmDraw[0]}
  [880] = {x=0.02, y=3.03, z=1, rx=90, ry=89.37, fatherId=FrmDraw[0]}
  [881] = {x=0.02, y=3.23, z=1, rx=90, ry=89.33, fatherId=FrmDraw[0]}
  [882] = {x=0.02, y=3.43, z=1, rx=90, ry=89.29, fatherId=FrmDraw[0]}
  [883] = {x=0.02, y=3.63, z=1, rx=90, ry=89.24, fatherId=FrmDraw[0]}
  [884] = {x=0.03, y=3.83, z=1, rx=90, ry=89.2, fatherId=FrmDraw[0]}
  [885] = {x=0.03, y=4.03, z=1, rx=90, ry=89.16, fatherId=FrmDraw[0]}
  [886] = {x=0.03, y=4.23, z=1, rx=90, ry=89.12, fatherId=FrmDraw[0]}
  [887] = {x=0.04, y=4.43, z=1, rx=90, ry=89.08, fatherId=FrmDraw[0]}
  [888] = {x=0.04, y=4.63, z=1, rx=90, ry=89.04, fatherId=FrmDraw[0]}
  [889] = {x=0.04, y=4.83, z=1, rx=90, ry=88.99, fatherId=FrmDraw[0]}
  [890] = {x=0.05, y=5.03, z=1, rx=90, ry=88.95, fatherId=FrmDraw[0]}
  [891] = {x=0.05, y=5.23, z=1, rx=90, ry=88.91, fatherId=FrmDraw[0]}
  [892] = {x=0.05, y=5.43, z=1, rx=90, ry=88.87, fatherId=FrmDraw[0]}
  [893] = {x=0.06, y=5.63, z=1, rx=90, ry=88.83, fatherId=FrmDraw[0]}
  [894] = {x=0.06, y=5.83, z=1, rx=90, ry=88.79, fatherId=FrmDraw[0]}
  [895] = {x=0.07, y=6.03, z=1, rx=90, ry=88.74, fatherId=FrmDraw[0]}
  [896] = {x=0.07, y=6.23, z=1, rx=90, ry=88.7, fatherId=FrmDraw[0]}
  [897] = {x=0.08, y=6.43, z=1, rx=90, ry=88.66, fatherId=FrmDraw[0]}
  [898] = {x=0.08, y=6.63, z=1, rx=90, ry=88.62, fatherId=FrmDraw[0]}
  [899] = {x=0.08, y=6.83, z=1, rx=90, ry=88.58, fatherId=FrmDraw[0]}
  [900] = {x=0.09, y=7.03, z=1, rx=90, ry=88.54, fatherId=FrmDraw[0]}
  [901] = {x=0.1, y=7.23, z=1, rx=90, ry=88.49, fatherId=FrmDraw[0]}
  [902] = {x=0.1, y=7.43, z=1, rx=90, ry=88.45, fatherId=FrmDraw[0]}
  [903] = {x=0.11, y=7.63, z=1, rx=90, ry=88.41, fatherId=FrmDraw[0]}
  [904] = {x=0.11, y=7.83, z=1, rx=90, ry=88.37, fatherId=FrmDraw[0]}
  [905] = {x=0.12, y=8.03, z=1, rx=90, ry=88.33, fatherId=FrmDraw[0]}
  [906] = {x=0.12, y=8.23, z=1, rx=90, ry=88.29, fatherId=FrmDraw[0]}
  [907] = {x=0.13, y=8.43, z=1, rx=90, ry=88.24, fatherId=FrmDraw[0]}
  [908] = {x=0.14, y=8.63, z=1, rx=90, ry=88.2, fatherId=FrmDraw[0]}
  [909] = {x=0.14, y=8.83, z=1, rx=90, ry=88.16, fatherId=FrmDraw[0]}
  [910] = {x=0.15, y=9.03, z=1, rx=90, ry=88.12, fatherId=FrmDraw[0]}
  [911] = {x=0.15, y=9.23, z=1, rx=90, ry=88.08, fatherId=FrmDraw[0]}
  [912] = {x=0.16, y=9.43, z=1, rx=90, ry=88.04, fatherId=FrmDraw[0]}
  [913] = {x=0.17, y=9.63, z=1, rx=90, ry=87.99, fatherId=FrmDraw[0]}
  [914] = {x=0.18, y=9.83, z=1, rx=90, ry=87.95, fatherId=FrmDraw[0]}
  [915] = {x=0.18, y=10.03, z=1, rx=90, ry=87.91, fatherId=FrmDraw[0]}
  [916] = {x=0.19, y=10.23, z=1, rx=90, ry=87.87, fatherId=FrmDraw[0]}
  [917] = {x=0.2, y=10.43, z=1, rx=90, ry=87.83, fatherId=FrmDraw[0]}
  [918] = {x=0.21, y=10.63, z=1, rx=90, ry=87.79, fatherId=FrmDraw[0]}
  [919] = {x=0.21, y=10.83, z=1, rx=90, ry=87.74, fatherId=FrmDraw[0]}
  [920] = {x=0.22, y=11.03, z=1, rx=90, ry=87.7, fatherId=FrmDraw[0]}
  [921] = {x=0.23, y=11.23, z=1, rx=90, ry=87.66, fatherId=FrmDraw[0]}
  [922] = {x=0.24, y=11.43, z=1, rx=90, ry=87.62, fatherId=FrmDraw[0]}
  [923] = {x=0.25, y=11.63, z=1, rx=90, ry=87.58, fatherId=FrmDraw[0]}
  [924] = {x=0.25, y=11.83, z=1, rx=90, ry=87.53, fatherId=FrmDraw[0]}
  [925] = {x=0.26, y=12.03, z=1, rx=90, ry=87.49, fatherId=FrmDraw[0]}
  [926] = {x=0.27, y=12.23, z=1, rx=90, ry=87.45, fatherId=FrmDraw[0]}
  [927] = {x=0.28, y=12.43, z=1, rx=90, ry=87.41, fatherId=FrmDraw[0]}
  [928] = {x=0.29, y=12.63, z=1, rx=90, ry=87.37, fatherId=FrmDraw[0]}
  [929] = {x=0.3, y=12.83, z=1, rx=90, ry=87.33, fatherId=FrmDraw[0]}
  [930] = {x=0.31, y=13.03, z=1, rx=90, ry=87.28, fatherId=FrmDraw[0]}
  [931] = {x=0.32, y=13.23, z=1, rx=90, ry=87.24, fatherId=FrmDraw[0]}
  [932] = {x=0.33, y=13.43, z=1, rx=90, ry=87.2, fatherId=FrmDraw[0]}
  [933] = {x=0.34, y=13.63, z=1, rx=90, ry=87.16, fatherId=FrmDraw[0]}
  [934] = {x=0.35, y=13.83, z=1, rx=90, ry=87.12, fatherId=FrmDraw[0]}
  [935] = {x=0.36, y=14.02, z=1, rx=90, ry=87.08, fatherId=FrmDraw[0]}
  [936] = {x=0.37, y=14.22, z=1, rx=90, ry=87.03, fatherId=FrmDraw[0]}
  [937] = {x=0.38, y=14.42, z=1, rx=90, ry=86.99, fatherId=FrmDraw[0]}
  [938] = {x=0.39, y=14.62, z=1, rx=90, ry=86.95, fatherId=FrmDraw[0]}
  [939] = {x=0.4, y=14.82, z=1, rx=90, ry=86.91, fatherId=FrmDraw[0]}
  [940] = {x=0.41, y=15.02, z=1, rx=90, ry=86.87, fatherId=FrmDraw[0]}
  [941] = {x=0.42, y=15.22, z=1, rx=90, ry=86.83, fatherId=FrmDraw[0]}
  [942] = {x=0.43, y=15.42, z=1, rx=90, ry=86.78, fatherId=FrmDraw[0]}
  [943] = {x=0.44, y=15.62, z=1, rx=90, ry=86.74, fatherId=FrmDraw[0]}
  [944] = {x=0.46, y=15.82, z=1, rx=90, ry=86.7, fatherId=FrmDraw[0]}
  [945] = {x=0.47, y=16.02, z=1, rx=90, ry=86.66, fatherId=FrmDraw[0]}
  [946] = {x=0.48, y=16.22, z=1, rx=90, ry=86.62, fatherId=FrmDraw[0]}
  [947] = {x=0.49, y=16.42, z=1, rx=90, ry=86.58, fatherId=FrmDraw[0]}
  [948] = {x=0.5, y=16.62, z=1, rx=90, ry=86.53, fatherId=FrmDraw[0]}
  [949] = {x=0.51, y=16.82, z=1, rx=90, ry=86.49, fatherId=FrmDraw[0]}
  [950] = {x=0.53, y=17.02, z=1, rx=90, ry=86.45, fatherId=FrmDraw[0]}
  [951] = {x=0.54, y=17.22, z=1, rx=90, ry=86.41, fatherId=FrmDraw[0]}
  [952] = {x=0.55, y=17.42, z=1, rx=90, ry=86.37, fatherId=FrmDraw[0]}
  [953] = {x=0.56, y=17.62, z=1, rx=90, ry=86.33, fatherId=FrmDraw[0]}
  [954] = {x=0.58, y=17.82, z=1, rx=90, ry=86.28, fatherId=FrmDraw[0]}
  [955] = {x=0.59, y=18.02, z=1, rx=90, ry=86.24, fatherId=FrmDraw[0]}
  [956] = {x=0.6, y=18.22, z=1, rx=90, ry=86.2, fatherId=FrmDraw[0]}
  [957] = {x=0.62, y=18.42, z=1, rx=90, ry=86.16, fatherId=FrmDraw[0]}
  [958] = {x=0.63, y=18.62, z=1, rx=90, ry=86.12, fatherId=FrmDraw[0]}
  [959] = {x=0.64, y=18.82, z=1, rx=90, ry=86.08, fatherId=FrmDraw[0]}
  [960] = {x=0.66, y=19.02, z=1, rx=90, ry=86.03, fatherId=FrmDraw[0]}
  [961] = {x=0.67, y=19.22, z=1, rx=90, ry=85.99, fatherId=FrmDraw[0]}
  [962] = {x=0.69, y=19.41, z=1, rx=90, ry=85.95, fatherId=FrmDraw[0]}
  [963] = {x=0.7, y=19.61, z=1, rx=90, ry=85.91, fatherId=FrmDraw[0]}
  [964] = {x=0.71, y=19.81, z=1, rx=90, ry=85.87, fatherId=FrmDraw[0]}
  [965] = {x=0.73, y=20.01, z=1, rx=90, ry=85.83, fatherId=FrmDraw[0]}
  [966] = {x=0.74, y=20.21, z=1, rx=90, ry=85.78, fatherId=FrmDraw[0]}
  [967] = {x=0.76, y=20.41, z=1, rx=90, ry=85.74, fatherId=FrmDraw[0]}
  [968] = {x=0.77, y=20.61, z=1, rx=90, ry=85.7, fatherId=FrmDraw[0]}
  [969] = {x=0.79, y=20.81, z=1, rx=90, ry=85.66, fatherId=FrmDraw[0]}
  [970] = {x=0.8, y=21.01, z=1, rx=90, ry=85.62, fatherId=FrmDraw[0]}
  [971] = {x=0.82, y=21.21, z=1, rx=90, ry=85.58, fatherId=FrmDraw[0]}
  [972] = {x=0.83, y=21.41, z=1, rx=90, ry=85.53, fatherId=FrmDraw[0]}
  [973] = {x=0.85, y=21.61, z=1, rx=90, ry=85.49, fatherId=FrmDraw[0]}
  [974] = {x=0.87, y=21.81, z=1, rx=90, ry=85.45, fatherId=FrmDraw[0]}
  [975] = {x=0.88, y=22.01, z=1, rx=90, ry=85.41, fatherId=FrmDraw[0]}
  [976] = {x=0.9, y=22.21, z=1, rx=90, ry=85.37, fatherId=FrmDraw[0]}
  [977] = {x=0.91, y=22.41, z=1, rx=90, ry=85.33, fatherId=FrmDraw[0]}
  [978] = {x=0.93, y=22.61, z=1, rx=90, ry=85.28, fatherId=FrmDraw[0]}
  [979] = {x=0.95, y=22.8, z=1, rx=90, ry=85.24, fatherId=FrmDraw[0]}
  [980] = {x=0.96, y=23, z=1, rx=90, ry=85.2, fatherId=FrmDraw[0]}
  [981] = {x=0.98, y=23.2, z=1, rx=90, ry=85.16, fatherId=FrmDraw[0]}
  [982] = {x=1, y=23.4, z=1, rx=90, ry=85.12, fatherId=FrmDraw[0]}
  [983] = {x=1.01, y=23.6, z=1, rx=90, ry=85.08, fatherId=FrmDraw[0]}
  [984] = {x=1.03, y=23.8, z=1, rx=90, ry=85.03, fatherId=FrmDraw[0]}
  [985] = {x=1.05, y=24, z=1, rx=90, ry=84.99, fatherId=FrmDraw[0]}
  [986] = {x=1.07, y=24.2, z=1, rx=90, ry=84.95, fatherId=FrmDraw[0]}
  [987] = {x=1.08, y=24.4, z=1, rx=90, ry=84.91, fatherId=FrmDraw[0]}
  [988] = {x=1.1, y=24.6, z=1, rx=90, ry=84.87, fatherId=FrmDraw[0]}
  [989] = {x=1.12, y=24.8, z=1, rx=90, ry=84.83, fatherId=FrmDraw[0]}
  [990] = {x=1.14, y=25, z=1, rx=90, ry=84.78, fatherId=FrmDraw[0]}
  [991] = {x=1.16, y=25.2, z=1, rx=90, ry=84.74, fatherId=FrmDraw[0]}
  [992] = {x=1.18, y=25.39, z=1, rx=90, ry=84.7, fatherId=FrmDraw[0]}
  [993] = {x=1.19, y=25.59, z=1, rx=90, ry=84.66, fatherId=FrmDraw[0]}
  [994] = {x=1.21, y=25.79, z=1, rx=90, ry=84.62, fatherId=FrmDraw[0]}
  [995] = {x=1.23, y=25.99, z=1, rx=90, ry=84.58, fatherId=FrmDraw[0]}
  [996] = {x=1.25, y=26.19, z=1, rx=90, ry=84.53, fatherId=FrmDraw[0]}
  [997] = {x=1.27, y=26.39, z=1, rx=90, ry=84.49, fatherId=FrmDraw[0]}
  [998] = {x=1.29, y=26.59, z=1, rx=90, ry=84.45, fatherId=FrmDraw[0]}
  [999] = {x=1.31, y=26.79, z=1, rx=90, ry=84.41, fatherId=FrmDraw[0]}
pointRx zero = {ry=90, rz=-3.944843}
public sio socket = {link=Socket\socket1}
string CmdBuffer[20]
string dataSend2PC = "(010010)"
string datar
string sScrPts = "OK"
string sString[1500]
  [0] = "52.63,-161.79,1.00,-90.00,-53.98,0.00,1,"
  [1] = "52.51,-161.63,1.00,-90.00,-54.00,0.00,0,"
  [2] = "52.39,-161.46,1.00,-90.00,-54.05,0.00,1,"
  [3] = "52.27,-161.30,1.00,-90.00,-54.09,0.00,0,"
  [4] = "52.16,-161.14,1.00,-90.00,-54.13,0.00,1,"
  [5] = "52.04,-160.98,1.00,-90.00,-54.17,0.00,0,"
  [6] = "51.92,-160.82,1.00,-90.00,-54.21,0.00,1,"
  [7] = "51.81,-160.65,1.00,-90.00,-54.25,0.00,0,"
  [8] = "51.69,-160.49,1.00,-90.00,-54.30,0.00,1,"
  [9] = "51.57,-160.33,1.00,-90.00,-54.34,0.00,0,"
  [10] = "51.46,-160.17,1.00,-90.00,-54.38,0.00,1,"
  [11] = "51.34,-160.00,1.00,-90.00,-54.42,0.00,0,"
  [12] = "51.22,-159.84,1.00,-90.00,-54.46,0.00,1,"
  [13] = "51.11,-159.68,1.00,-90.00,-54.50,0.00,0,"
  [14] = "50.99,-159.52,1.00,-90.00,-54.55,0.00,1,"
  [15] = "50.88,-159.35,1.00,-90.00,-54.59,0.00,0,"
  [16] = "50.76,-159.19,1.00,-90.00,-54.63,0.00,1,"
  [17] = "50.64,-159.03,1.00,-90.00,-54.67,0.00,0,"
  [18] = "50.53,-158.86,1.00,-90.00,-54.71,0.00,1,"
  [19] = "50.41,-158.70,1.00,-90.00,-54.75,0.00,0,"
  [20] = "50.30,-158.54,1.00,-90.00,-54.80,0.00,1,"
  [21] = "50.18,-158.37,1.00,-90.00,-54.84,0.00,0,"
  [22] = "50.07,-158.21,1.00,-90.00,-54.88,0.00,1,"
  [23] = "49.95,-158.05,1.00,-90.00,-54.92,0.00,0,"
  [24] = "49.84,-157.88,1.00,-90.00,-54.96,0.00,1,"
  [25] = "49.72,-157.72,1.00,-90.00,-55.00,0.00,0,"
  [26] = "49.61,-157.55,1.00,-90.00,-55.05,0.00,1,"
  [27] = "49.49,-157.39,1.00,-90.00,-55.09,0.00,0,"
  [28] = "49.38,-157.23,1.00,-90.00,-55.13,0.00,1,"
  [29] = "49.26,-157.06,1.00,-90.00,-55.17,0.00,0,"
  [30] = "49.15,-156.90,1.00,-90.00,-55.21,0.00,1,"
  [31] = "49.04,-156.73,1.00,-90.00,-55.25,0.00,0,"
  [32] = "48.92,-156.57,1.00,-90.00,-55.30,0.00,1,"
  [33] = "48.81,-156.40,1.00,-90.00,-55.34,0.00,0,"
  [34] = "48.69,-156.24,1.00,-90.00,-55.38,0.00,1,"
  [35] = "48.58,-156.08,1.00,-90.00,-55.42,0.00,0,"
  [36] = "48.47,-155.91,1.00,-90.00,-55.46,0.00,1,"
  [37] = "48.35,-155.75,1.00,-90.00,-55.50,0.00,0,"
  [38] = "48.24,-155.58,1.00,-90.00,-55.55,0.00,1,"
  [39] = "48.13,-155.42,1.00,-90.00,-55.59,0.00,0,"
  [40] = "48.02,-155.25,1.00,-90.00,-55.63,0.00,1,"
  [41] = "47.90,-155.09,1.00,-90.00,-55.67,0.00,0,"
  [42] = "47.79,-154.92,1.00,-90.00,-55.71,0.00,1,"
  [43] = "47.68,-154.76,1.00,-90.00,-55.75,0.00,0,"
  [44] = "47.56,-154.59,1.00,-90.00,-55.80,0.00,1,"
  [45] = "47.45,-154.42,1.00,-90.00,-55.84,0.00,0,"
  [46] = "47.34,-154.26,1.00,-90.00,-55.88,0.00,1,"
  [47] = "47.23,-154.09,1.00,-90.00,-55.92,0.00,0,"
  [48] = "47.12,-153.93,1.00,-90.00,-55.96,0.00,1,"
  [49] = "47.00,-153.76,1.00,-90.00,-56.00,0.00,0,"
  [50] = "46.89,-153.60,1.00,-90.00,-56.05,0.00,1,"
  [51] = "46.78,-153.43,1.00,-90.00,-56.09,0.00,0,"
  [52] = "46.67,-153.26,1.00,-90.00,-56.13,0.00,1,"
  [53] = "46.56,-153.10,1.00,-90.00,-56.17,0.00,0,"
  [54] = "46.45,-152.93,1.00,-90.00,-56.21,0.00,1,"
  [55] = "46.34,-152.77,1.00,-90.00,-56.25,0.00,0,"
  [56] = "46.22,-152.60,1.00,-90.00,-56.30,0.00,1,"
  [57] = "46.11,-152.43,1.00,-90.00,-56.34,0.00,0,"
  [58] = "46.00,-152.27,1.00,-90.00,-56.38,0.00,1,"
  [59] = "45.89,-152.10,1.00,-90.00,-56.42,0.00,0,"
  [60] = "45.78,-151.93,1.00,-90.00,-56.46,0.00,1,"
  [61] = "45.67,-151.77,1.00,-90.00,-56.50,0.00,0,"
  [62] = "45.56,-151.60,1.00,-90.00,-56.55,0.00,1,"
  [63] = "45.45,-151.43,1.00,-90.00,-56.59,0.00,0,"
  [64] = "45.34,-151.27,1.00,-90.00,-56.63,0.00,1,"
  [65] = "45.23,-151.10,1.00,-90.00,-56.67,0.00,0,"
  [66] = "45.12,-150.93,1.00,-90.00,-56.71,0.00,1,"
  [67] = "45.01,-150.76,1.00,-90.00,-56.75,0.00,0,"
  [68] = "44.90,-150.60,1.00,-90.00,-56.80,0.00,1,"
  [69] = "44.79,-150.43,1.00,-90.00,-56.84,0.00,0,"
  [70] = "44.68,-150.26,1.00,-90.00,-56.88,0.00,1,"
  [71] = "44.57,-150.09,1.00,-90.00,-56.92,0.00,0,"
  [72] = "44.46,-149.93,1.00,-90.00,-56.96,0.00,1,"
  [73] = "44.35,-149.76,1.00,-90.00,-57.00,0.00,0,"
  [74] = "44.25,-149.59,1.00,-90.00,-57.05,0.00,1,"
  [75] = "44.14,-149.42,1.00,-90.00,-57.09,0.00,0,"
  [76] = "44.03,-149.26,1.00,-90.00,-57.13,0.00,1,"
  [77] = "43.92,-149.09,1.00,-90.00,-57.17,0.00,0,"
  [78] = "43.81,-148.92,1.00,-90.00,-57.21,0.00,1,"
  [79] = "43.70,-148.75,1.00,-90.00,-57.25,0.00,0,"
  [80] = "43.60,-148.58,1.00,-90.00,-57.30,0.00,1,"
  [81] = "43.49,-148.41,1.00,-90.00,-57.34,0.00,0,"
  [82] = "43.38,-148.25,1.00,-90.00,-57.38,0.00,1,"
  [83] = "43.27,-148.08,1.00,-90.00,-57.42,0.00,0,"
  [84] = "43.16,-147.91,1.00,-90.00,-57.46,0.00,1,"
  [85] = "43.06,-147.74,1.00,-90.00,-57.50,0.00,0,"
  [86] = "42.95,-147.57,1.00,-90.00,-57.55,0.00,1,"
  [87] = "42.84,-147.40,1.00,-90.00,-57.59,0.00,0,"
  [88] = "42.73,-147.23,1.00,-90.00,-57.63,0.00,1,"
  [89] = "42.63,-147.07,1.00,-90.00,-57.67,0.00,0,"
  [90] = "42.52,-146.90,1.00,-90.00,-57.71,0.00,1,"
  [91] = "42.41,-146.73,1.00,-90.00,-57.75,0.00,0,"
  [92] = "42.31,-146.56,1.00,-90.00,-57.80,0.00,1,"
  [93] = "42.20,-146.39,1.00,-90.00,-57.84,0.00,0,"
  [94] = "42.09,-146.22,1.00,-90.00,-57.88,0.00,1,"
  [95] = "41.99,-146.05,1.00,-90.00,-57.92,0.00,0,"
  [96] = "41.88,-145.88,1.00,-90.00,-57.96,0.00,1,"
  [97] = "41.78,-145.71,1.00,-90.00,-58.00,0.00,0,"
  [98] = "41.67,-145.54,1.00,-90.00,-58.05,0.00,1,"
  [99] = "41.56,-145.37,1.00,-90.00,-58.09,0.00,0,"
  [100] = "41.46,-145.20,1.00,-90.00,-58.13,0.00,1,"
  [101] = "41.35,-145.03,1.00,-90.00,-58.17,0.00,0,"
  [102] = "41.25,-144.86,1.00,-90.00,-58.21,0.00,1,"
  [103] = "41.14,-144.69,1.00,-90.00,-58.25,0.00,0,"
  [104] = "41.04,-144.52,1.00,-90.00,-58.30,0.00,1,"
  [105] = "40.93,-144.35,1.00,-90.00,-58.34,0.00,0,"
  [106] = "40.83,-144.18,1.00,-90.00,-58.38,0.00,1,"
  [107] = "40.72,-144.01,1.00,-90.00,-58.42,0.00,0,"
  [108] = "40.62,-143.84,1.00,-90.00,-58.46,0.00,1,"
  [109] = "40.51,-143.67,1.00,-90.00,-58.50,0.00,0,"
  [110] = "40.41,-143.50,1.00,-90.00,-58.55,0.00,1,"
  [111] = "40.30,-143.33,1.00,-90.00,-58.59,0.00,0,"
  [112] = "40.20,-143.16,1.00,-90.00,-58.63,0.00,1,"
  [113] = "40.10,-142.99,1.00,-90.00,-58.67,0.00,0,"
  [114] = "39.99,-142.82,1.00,-90.00,-58.71,0.00,1,"
  [115] = "39.89,-142.65,1.00,-90.00,-58.75,0.00,0,"
  [116] = "39.79,-142.47,1.00,-90.00,-58.80,0.00,1,"
  [117] = "39.68,-142.30,1.00,-90.00,-58.84,0.00,0,"
  [118] = "39.58,-142.13,1.00,-90.00,-58.88,0.00,1,"
  [119] = "39.47,-141.96,1.00,-90.00,-58.92,0.00,0,"
  [120] = "39.37,-141.79,1.00,-90.00,-58.96,0.00,1,"
  [121] = "39.27,-141.62,1.00,-90.00,-59.00,0.00,0,"
  [122] = "39.17,-141.45,1.00,-90.00,-59.05,0.00,1,"
  [123] = "39.06,-141.28,1.00,-90.00,-59.09,0.00,0,"
  [124] = "38.96,-141.10,1.00,-90.00,-59.13,0.00,1,"
  [125] = "38.86,-140.93,1.00,-90.00,-59.17,0.00,0,"
  [126] = "38.76,-140.76,1.00,-90.00,-59.21,0.00,1,"
  [127] = "38.65,-140.59,1.00,-90.00,-59.25,0.00,0,"
  [128] = "38.55,-140.42,1.00,-90.00,-59.30,0.00,1,"
  [129] = "38.45,-140.24,1.00,-90.00,-59.34,0.00,0,"
  [130] = "38.35,-140.07,1.00,-90.00,-59.38,0.00,1,"
  [131] = "38.24,-139.90,1.00,-90.00,-59.42,0.00,0,"
  [132] = "38.14,-139.73,1.00,-90.00,-59.46,0.00,1,"
  [133] = "38.04,-139.56,1.00,-90.00,-59.50,0.00,0,"
  [134] = "37.94,-139.38,1.00,-90.00,-59.55,0.00,1,"
  [135] = "37.84,-139.21,1.00,-90.00,-59.59,0.00,0,"
  [136] = "37.74,-139.04,1.00,-90.00,-59.63,0.00,1,"
  [137] = "37.64,-138.87,1.00,-90.00,-59.67,0.00,0,"
  [138] = "37.54,-138.69,1.00,-90.00,-59.71,0.00,1,"
  [139] = "37.43,-138.52,1.00,-90.00,-59.75,0.00,0,"
  [140] = "37.33,-138.35,1.00,-90.00,-59.80,0.00,1,"
  [141] = "37.23,-138.17,1.00,-90.00,-59.84,0.00,0,"
  [142] = "37.13,-138.00,1.00,-90.00,-59.88,0.00,1,"
  [143] = "37.03,-137.83,1.00,-90.00,-59.92,0.00,0,"
  [144] = "36.93,-137.66,1.00,-90.00,-59.96,0.00,1,"
  [145] = "36.83,-137.48,1.00,-90.00,-60.00,0.00,0,"
  [146] = "36.73,-137.31,1.00,-90.00,-60.05,0.00,1,"
  [147] = "36.63,-137.14,1.00,-90.00,-60.09,0.00,0,"
  [148] = "36.53,-136.96,1.00,-90.00,-60.13,0.00,1,"
  [149] = "36.43,-136.79,1.00,-90.00,-60.17,0.00,0,"
  [150] = "36.33,-136.62,1.00,-90.00,-60.21,0.00,1,"
  [151] = "36.24,-136.44,1.00,-90.00,-60.25,0.00,0,"
  [152] = "36.14,-136.27,1.00,-90.00,-60.30,0.00,1,"
  [153] = "36.04,-136.09,1.00,-90.00,-60.34,0.00,0,"
  [154] = "35.94,-135.92,1.00,-90.00,-60.38,0.00,1,"
  [155] = "35.84,-135.75,1.00,-90.00,-60.42,0.00,0,"
  [156] = "35.74,-135.57,1.00,-90.00,-60.46,0.00,1,"
  [157] = "35.64,-135.40,1.00,-90.00,-60.50,0.00,0,"
  [158] = "35.54,-135.22,1.00,-90.00,-60.55,0.00,1,"
  [159] = "35.45,-135.05,1.00,-90.00,-60.59,0.00,0,"
  [160] = "35.35,-134.88,1.00,-90.00,-60.63,0.00,1,"
  [161] = "35.25,-134.70,1.00,-90.00,-60.67,0.00,0,"
  [162] = "35.15,-134.53,1.00,-90.00,-60.71,0.00,1,"
  [163] = "35.05,-134.35,1.00,-90.00,-60.75,0.00,0,"
  [164] = "34.96,-134.18,1.00,-90.00,-60.80,0.00,1,"
  [165] = "34.86,-134.00,1.00,-90.00,-60.84,0.00,0,"
  [166] = "34.76,-133.83,1.00,-90.00,-60.88,0.00,1,"
  [167] = "34.66,-133.65,1.00,-90.00,-60.92,0.00,0,"
  [168] = "34.57,-133.48,1.00,-90.00,-60.96,0.00,1,"
  [169] = "34.47,-133.30,1.00,-90.00,-61.00,0.00,0,"
  [170] = "34.37,-133.13,1.00,-90.00,-61.05,0.00,1,"
  [171] = "34.28,-132.95,1.00,-90.00,-61.09,0.00,0,"
  [172] = "34.18,-132.78,1.00,-90.00,-61.13,0.00,1,"
  [173] = "34.08,-132.60,1.00,-90.00,-61.17,0.00,0,"
  [174] = "33.99,-132.43,1.00,-90.00,-61.21,0.00,1,"
  [175] = "33.89,-132.25,1.00,-90.00,-61.25,0.00,0,"
  [176] = "33.79,-132.08,1.00,-90.00,-61.30,0.00,1,"
  [177] = "33.70,-131.90,1.00,-90.00,-61.34,0.00,0,"
  [178] = "33.60,-131.73,1.00,-90.00,-61.38,0.00,1,"
  [179] = "33.51,-131.55,1.00,-90.00,-61.42,0.00,0,"
  [180] = "33.41,-131.38,1.00,-90.00,-61.46,0.00,1,"
  [181] = "33.32,-131.20,1.00,-90.00,-61.50,0.00,0,"
  [182] = "33.22,-131.02,1.00,-90.00,-61.55,0.00,1,"
  [183] = "33.12,-130.85,1.00,-90.00,-61.59,0.00,0,"
  [184] = "33.03,-130.67,1.00,-90.00,-61.63,0.00,1,"
  [185] = "32.93,-130.50,1.00,-90.00,-61.67,0.00,0,"
  [186] = "32.84,-130.32,1.00,-90.00,-61.71,0.00,1,"
  [187] = "32.74,-130.14,1.00,-90.00,-61.75,0.00,0,"
  [188] = "32.65,-129.97,1.00,-90.00,-61.80,0.00,1,"
  [189] = "32.56,-129.79,1.00,-90.00,-61.84,0.00,0,"
  [190] = "32.46,-129.62,1.00,-90.00,-61.88,0.00,1,"
  [191] = "32.37,-129.44,1.00,-90.00,-61.92,0.00,0,"
  [192] = "32.27,-129.26,1.00,-90.00,-61.96,0.00,1,"
  [193] = "32.18,-129.09,1.00,-90.00,-62.00,0.00,0,"
  [194] = "32.09,-128.91,1.00,-90.00,-62.05,0.00,1,"
  [195] = "31.99,-128.73,1.00,-90.00,-62.09,0.00,0,"
  [196] = "31.90,-128.56,1.00,-90.00,-62.13,0.00,1,"
  [197] = "31.80,-128.38,1.00,-90.00,-62.17,0.00,0,"
  [198] = "31.71,-128.20,1.00,-90.00,-62.21,0.00,1,"
  [199] = "31.62,-128.03,1.00,-90.00,-62.25,0.00,0,"
  [200] = "31.53,-127.85,1.00,-90.00,-62.30,0.00,1,"
  [201] = "31.43,-127.67,1.00,-90.00,-62.34,0.00,0,"
  [202] = "31.34,-127.49,1.00,-90.00,-62.38,0.00,1,"
  [203] = "31.25,-127.32,1.00,-90.00,-62.42,0.00,0,"
  [204] = "31.15,-127.14,1.00,-90.00,-62.46,0.00,1,"
  [205] = "31.06,-126.96,1.00,-90.00,-62.50,0.00,0,"
  [206] = "30.97,-126.78,1.00,-90.00,-62.55,0.00,1,"
  [207] = "30.88,-126.61,1.00,-90.00,-62.59,0.00,0,"
  [208] = "30.79,-126.43,1.00,-90.00,-62.63,0.00,1,"
  [209] = "30.69,-126.25,1.00,-90.00,-62.67,0.00,0,"
  [210] = "30.60,-126.07,1.00,-90.00,-62.71,0.00,1,"
  [211] = "30.51,-125.90,1.00,-90.00,-62.75,0.00,0,"
  [212] = "30.42,-125.72,1.00,-90.00,-62.80,0.00,1,"
  [213] = "30.33,-125.54,1.00,-90.00,-62.84,0.00,0,"
  [214] = "30.24,-125.36,1.00,-90.00,-62.88,0.00,1,"
  [215] = "30.15,-125.18,1.00,-90.00,-62.92,0.00,0,"
  [216] = "30.05,-125.01,1.00,-90.00,-62.96,0.00,1,"
  [217] = "29.96,-124.83,1.00,-90.00,-63.00,0.00,0,"
  [218] = "29.87,-124.65,1.00,-90.00,-63.05,0.00,1,"
  [219] = "29.78,-124.47,1.00,-90.00,-63.09,0.00,0,"
  [220] = "29.69,-124.29,1.00,-90.00,-63.13,0.00,1,"
  [221] = "29.60,-124.11,1.00,-90.00,-63.17,0.00,0,"
  [222] = "29.51,-123.94,1.00,-90.00,-63.21,0.00,1,"
  [223] = "29.42,-123.76,1.00,-90.00,-63.25,0.00,0,"
  [224] = "29.33,-123.58,1.00,-90.00,-63.30,0.00,1,"
  [225] = "29.24,-123.40,1.00,-90.00,-63.34,0.00,0,"
  [226] = "29.15,-123.22,1.00,-90.00,-63.38,0.00,1,"
  [227] = "29.06,-123.04,1.00,-90.00,-63.42,0.00,0,"
  [228] = "28.97,-122.86,1.00,-90.00,-63.46,0.00,1,"
  [229] = "28.88,-122.68,1.00,-90.00,-63.50,0.00,0,"
  [230] = "28.79,-122.51,1.00,-90.00,-63.55,0.00,1,"
  [231] = "28.71,-122.33,1.00,-90.00,-63.59,0.00,0,"
  [232] = "28.62,-122.15,1.00,-90.00,-63.63,0.00,1,"
  [233] = "28.53,-121.97,1.00,-90.00,-63.67,0.00,0,"
  [234] = "28.44,-121.79,1.00,-90.00,-63.71,0.00,1,"
  [235] = "28.35,-121.61,1.00,-90.00,-63.75,0.00,0,"
  [236] = "28.26,-121.43,1.00,-90.00,-63.80,0.00,1,"
  [237] = "28.17,-121.25,1.00,-90.00,-63.84,0.00,0,"
  [238] = "28.09,-121.07,1.00,-90.00,-63.88,0.00,1,"
  [239] = "28.00,-120.89,1.00,-90.00,-63.92,0.00,0,"
  [240] = "27.91,-120.71,1.00,-90.00,-63.96,0.00,1,"
  [241] = "27.82,-120.53,1.00,-90.00,-64.00,0.00,0,"
  [242] = "27.73,-120.35,1.00,-90.00,-64.05,0.00,1,"
  [243] = "27.65,-120.17,1.00,-90.00,-64.09,0.00,0,"
  [244] = "27.56,-119.99,1.00,-90.00,-64.13,0.00,1,"
  [245] = "27.47,-119.81,1.00,-90.00,-64.17,0.00,0,"
  [246] = "27.39,-119.63,1.00,-90.00,-64.21,0.00,1,"
  [247] = "27.30,-119.45,1.00,-90.00,-64.25,0.00,0,"
  [248] = "27.21,-119.27,1.00,-90.00,-64.30,0.00,1,"
  [249] = "27.12,-119.09,1.00,-90.00,-64.34,0.00,0,"
  [250] = "27.04,-118.91,1.00,-90.00,-64.38,0.00,1,"
  [251] = "26.95,-118.73,1.00,-90.00,-64.42,0.00,0,"
  [252] = "26.87,-118.55,1.00,-90.00,-64.46,0.00,1,"
  [253] = "26.78,-118.37,1.00,-90.00,-64.50,0.00,0,"
  [254] = "26.69,-118.19,1.00,-90.00,-64.55,0.00,1,"
  [255] = "26.61,-118.01,1.00,-90.00,-64.59,0.00,0,"
  [256] = "26.52,-117.83,1.00,-90.00,-64.63,0.00,1,"
  [257] = "26.44,-117.65,1.00,-90.00,-64.67,0.00,0,"
  [258] = "26.35,-117.47,1.00,-90.00,-64.71,0.00,1,"
  [259] = "26.27,-117.29,1.00,-90.00,-64.75,0.00,0,"
  [260] = "26.18,-117.11,1.00,-90.00,-64.80,0.00,1,"
  [261] = "26.09,-116.92,1.00,-90.00,-64.84,0.00,0,"
  [262] = "26.01,-116.74,1.00,-90.00,-64.88,0.00,1,"
  [263] = "25.93,-116.56,1.00,-90.00,-64.92,0.00,0,"
  [264] = "25.84,-116.38,1.00,-90.00,-64.96,0.00,1,"
  [265] = "25.76,-116.20,1.00,-90.00,-65.00,0.00,0,"
  [266] = "25.67,-116.02,1.00,-90.00,-65.05,0.00,1,"
  [267] = "25.59,-115.84,1.00,-90.00,-65.09,0.00,0,"
  [268] = "25.50,-115.66,1.00,-90.00,-65.13,0.00,1,"
  [269] = "25.42,-115.47,1.00,-90.00,-65.17,0.00,0,"
  [270] = "25.33,-115.29,1.00,-90.00,-65.21,0.00,1,"
  [271] = "25.25,-115.11,1.00,-90.00,-65.25,0.00,0,"
  [272] = "25.17,-114.93,1.00,-90.00,-65.30,0.00,1,"
  [273] = "25.08,-114.75,1.00,-90.00,-65.34,0.00,0,"
  [274] = "25.00,-114.57,1.00,-90.00,-65.38,0.00,1,"
  [275] = "24.92,-114.38,1.00,-90.00,-65.42,0.00,0,"
  [276] = "24.83,-114.20,1.00,-90.00,-65.46,0.00,1,"
  [277] = "24.75,-114.02,1.00,-90.00,-65.50,0.00,0,"
  [278] = "24.67,-113.84,1.00,-90.00,-65.55,0.00,1,"
  [279] = "24.59,-113.66,1.00,-90.00,-65.59,0.00,0,"
  [280] = "24.50,-113.47,1.00,-90.00,-65.63,0.00,1,"
  [281] = "24.42,-113.29,1.00,-90.00,-65.67,0.00,0,"
  [282] = "24.34,-113.11,1.00,-90.00,-65.71,0.00,1,"
  [283] = "24.26,-112.93,1.00,-90.00,-65.75,0.00,0,"
  [284] = "24.17,-112.74,1.00,-90.00,-65.80,0.00,1,"
  [285] = "24.09,-112.56,1.00,-90.00,-65.84,0.00,0,"
  [286] = "24.01,-112.38,1.00,-90.00,-65.88,0.00,1,"
  [287] = "23.93,-112.20,1.00,-90.00,-65.92,0.00,0,"
  [288] = "23.85,-112.01,1.00,-90.00,-65.96,0.00,1,"
  [289] = "23.77,-111.83,1.00,-90.00,-66.00,0.00,0,"
  [290] = "23.68,-111.65,1.00,-90.00,-66.05,0.00,1,"
  [291] = "23.60,-111.47,1.00,-90.00,-66.09,0.00,0,"
  [292] = "23.52,-111.28,1.00,-90.00,-66.13,0.00,1,"
  [293] = "23.44,-111.10,1.00,-90.00,-66.17,0.00,0,"
  [294] = "23.36,-110.92,1.00,-90.00,-66.21,0.00,1,"
  [295] = "23.28,-110.73,1.00,-90.00,-66.25,0.00,0,"
  [296] = "23.20,-110.55,1.00,-90.00,-66.30,0.00,1,"
  [297] = "23.12,-110.37,1.00,-90.00,-66.34,0.00,0,"
  [298] = "23.04,-110.18,1.00,-90.00,-66.38,0.00,1,"
  [299] = "22.96,-110.00,1.00,-90.00,-66.42,0.00,0,"
  [300] = "22.88,-109.82,1.00,-90.00,-66.46,0.00,1,"
  [301] = "22.80,-109.63,1.00,-90.00,-66.50,0.00,0,"
  [302] = "22.72,-109.45,1.00,-90.00,-66.55,0.00,1,"
  [303] = "22.64,-109.27,1.00,-90.00,-66.59,0.00,0,"
  [304] = "22.56,-109.08,1.00,-90.00,-66.63,0.00,1,"
  [305] = "22.48,-108.90,1.00,-90.00,-66.67,0.00,0,"
  [306] = "22.40,-108.72,1.00,-90.00,-66.71,0.00,1,"
  [307] = "22.32,-108.53,1.00,-90.00,-66.75,0.00,0,"
  [308] = "22.24,-108.35,1.00,-90.00,-66.80,0.00,1,"
  [309] = "22.17,-108.17,1.00,-90.00,-66.84,0.00,0,"
  [310] = "22.09,-107.98,1.00,-90.00,-66.88,0.00,1,"
  [311] = "22.01,-107.80,1.00,-90.00,-66.92,0.00,0,"
  [312] = "21.93,-107.61,1.00,-90.00,-66.96,0.00,1,"
  [313] = "21.85,-107.43,1.00,-90.00,-67.00,0.00,0,"
  [314] = "21.77,-107.25,1.00,-90.00,-67.05,0.00,1,"
  [315] = "21.70,-107.06,1.00,-90.00,-67.09,0.00,0,"
  [316] = "21.62,-106.88,1.00,-90.00,-67.13,0.00,1,"
  [317] = "21.54,-106.69,1.00,-90.00,-67.17,0.00,0,"
  [318] = "21.46,-106.51,1.00,-90.00,-67.21,0.00,1,"
  [319] = "21.39,-106.32,1.00,-90.00,-67.25,0.00,0,"
  [320] = "21.31,-106.14,1.00,-90.00,-67.30,0.00,1,"
  [321] = "21.23,-105.96,1.00,-90.00,-67.34,0.00,0,"
  [322] = "21.15,-105.77,1.00,-90.00,-67.38,0.00,1,"
  [323] = "21.08,-105.59,1.00,-90.00,-67.42,0.00,0,"
  [324] = "21.00,-105.40,1.00,-90.00,-67.46,0.00,1,"
  [325] = "20.92,-105.22,1.00,-90.00,-67.50,0.00,0,"
  [326] = "20.85,-105.03,1.00,-90.00,-67.55,0.00,1,"
  [327] = "20.77,-104.85,1.00,-90.00,-67.59,0.00,0,"
  [328] = "20.70,-104.66,1.00,-90.00,-67.63,0.00,1,"
  [329] = "20.62,-104.48,1.00,-90.00,-67.67,0.00,0,"
  [330] = "20.54,-104.29,1.00,-90.00,-67.71,0.00,1,"
  [331] = "20.47,-104.11,1.00,-90.00,-67.75,0.00,0,"
  [332] = "20.39,-103.92,1.00,-90.00,-67.80,0.00,1,"
  [333] = "20.32,-103.74,1.00,-90.00,-67.84,0.00,0,"
  [334] = "20.24,-103.55,1.00,-90.00,-67.88,0.00,1,"
  [335] = "20.17,-103.37,1.00,-90.00,-67.92,0.00,0,"
  [336] = "20.09,-103.18,1.00,-90.00,-67.96,0.00,1,"
  [337] = "20.02,-103.00,1.00,-90.00,-68.00,0.00,0,"
  [338] = "19.94,-102.81,1.00,-90.00,-68.05,0.00,1,"
  [339] = "19.87,-102.62,1.00,-90.00,-68.09,0.00,0,"
  [340] = "19.79,-102.44,1.00,-90.00,-68.13,0.00,1,"
  [341] = "19.72,-102.25,1.00,-90.00,-68.17,0.00,0,"
  [342] = "19.64,-102.07,1.00,-90.00,-68.21,0.00,1,"
  [343] = "19.57,-101.88,1.00,-90.00,-68.25,0.00,0,"
  [344] = "19.49,-101.70,1.00,-90.00,-68.30,0.00,1,"
  [345] = "19.42,-101.51,1.00,-90.00,-68.34,0.00,0,"
  [346] = "19.35,-101.32,1.00,-90.00,-68.38,0.00,1,"
  [347] = "19.27,-101.14,1.00,-90.00,-68.42,0.00,0,"
  [348] = "19.20,-100.95,1.00,-90.00,-68.46,0.00,1,"
  [349] = "19.13,-100.77,1.00,-90.00,-68.50,0.00,0,"
  [350] = "19.05,-100.58,1.00,-90.00,-68.55,0.00,1,"
  [351] = "18.98,-100.39,1.00,-90.00,-68.59,0.00,0,"
  [352] = "18.91,-100.21,1.00,-90.00,-68.63,0.00,1,"
  [353] = "18.83,-100.02,1.00,-90.00,-68.67,0.00,0,"
  [354] = "18.76,-99.83,1.00,-90.00,-68.71,0.00,1,"
  [355] = "18.69,-99.65,1.00,-90.00,-68.75,0.00,0,"
  [356] = "18.62,-99.46,1.00,-90.00,-68.80,0.00,1,"
  [357] = "18.54,-99.28,1.00,-90.00,-68.84,0.00,0,"
  [358] = "18.47,-99.09,1.00,-90.00,-68.88,0.00,1,"
  [359] = "18.40,-98.90,1.00,-90.00,-68.92,0.00,0,"
  [360] = "18.33,-98.72,1.00,-90.00,-68.96,0.00,1,"
  [361] = "18.26,-98.53,1.00,-90.00,-69.00,0.00,0,"
  [362] = "18.19,-98.34,1.00,-90.00,-69.05,0.00,1,"
  [363] = "18.11,-98.16,1.00,-90.00,-69.09,0.00,0,"
  [364] = "18.04,-97.97,1.00,-90.00,-69.13,0.00,1,"
  [365] = "17.97,-97.78,1.00,-90.00,-69.17,0.00,0,"
